//     PlcTask Inputs/GVL_iXlinker.EtherCAT_Master_ERxxxx.Beckhoff_ER2xxx.Beckhoff_ER2xxxEK1122.A_0015_ER2038_0002_0018.Diag_Channel_4.Input <-> Diag Channel 4/Input
//     PlcTask Inputs/GVL_iXlinker.EtherCAT_Master_ERxxxx.Beckhoff_ER2xxx.Beckhoff_ER2xxxEK1122.A_0015_ER2038_0002_0018.Diag_Channel_5.Input <-> Diag Channel 5/Input
//     PlcTask Inputs/GVL_iXlinker.EtherCAT_Master_ERxxxx.Beckhoff_ER2xxx.Beckhoff_ER2xxxEK1122.A_0015_ER2038_0002_0018.Diag_Channel_6.Input <-> Diag Channel 6/Input
//     PlcTask Inputs/GVL_iXlinker.EtherCAT_Master_ERxxxx.Beckhoff_ER2xxx.Beckhoff_ER2xxxEK1122.A_0015_ER2038_0002_0018.Diag_Channel_7.Input <-> Diag Channel 7/Input
//     PlcTask Inputs/GVL_iXlinker.EtherCAT_Master_ERxxxx.Beckhoff_ER2xxx.Beckhoff_ER2xxxEK1122.A_0015_ER2038_0002_0018.Diag_Channel_8.Input <-> Diag Channel 8/Input
//     PlcTask Outputs/GVL_iXlinker.EtherCAT_Master_ERxxxx.Beckhoff_ER2xxx.Beckhoff_ER2xxxEK1122.A_0015_ER2038_0002_0018.Channel_1.Output <-> Channel 1/Output
//     PlcTask Outputs/GVL_iXlinker.EtherCAT_Master_ERxxxx.Beckhoff_ER2xxx.Beckhoff_ER2xxxEK1122.A_0015_ER2038_0002_0018.Channel_2.Output <-> Channel 2/Output
//     PlcTask Outputs/GVL_iXlinker.EtherCAT_Master_ERxxxx.Beckhoff_ER2xxx.Beckhoff_ER2xxxEK1122.A_0015_ER2038_0002_0018.Channel_3.Output <-> Channel 3/Output
//     PlcTask Outputs/GVL_iXlinker.EtherCAT_Master_ERxxxx.Beckhoff_ER2xxx.Beckhoff_ER2xxxEK1122.A_0015_ER2038_0002_0018.Channel_4.Output <-> Channel 4/Output
//     PlcTask Outputs/GVL_iXlinker.EtherCAT_Master_ERxxxx.Beckhoff_ER2xxx.Beckhoff_ER2xxxEK1122.A_0015_ER2038_0002_0018.Channel_5.Output <-> Channel 5/Output
//     PlcTask Outputs/GVL_iXlinker.EtherCAT_Master_ERxxxx.Beckhoff_ER2xxx.Beckhoff_ER2xxxEK1122.A_0015_ER2038_0002_0018.Channel_6.Output <-> Channel 6/Output
//     PlcTask Outputs/GVL_iXlinker.EtherCAT_Master_ERxxxx.Beckhoff_ER2xxx.Beckhoff_ER2xxxEK1122.A_0015_ER2038_0002_0018.Channel_7.Output <-> Channel 7/Output
//     PlcTask Outputs/GVL_iXlinker.EtherCAT_Master_ERxxxx.Beckhoff_ER2xxx.Beckhoff_ER2xxxEK1122.A_0015_ER2038_0002_0018.Channel_8.Output <-> Channel 8/Output
//     PlcTask Inputs/GVL_iXlinker.EtherCAT_Master_ERxxxx.Beckhoff_ER2xxx.Beckhoff_ER2xxxEK1122.A_0015_ER2038_0002_0018.WcState.WcState <-> WcState/WcState
//     PlcTask Inputs/GVL_iXlinker.EtherCAT_Master_ERxxxx.Beckhoff_ER2xxx.Beckhoff_ER2xxxEK1122.A_0015_ER2038_0002_0018.WcState.InputToggle <-> WcState/InputToggle
//     PlcTask Inputs/GVL_iXlinker.EtherCAT_Master_ERxxxx.Beckhoff_ER2xxx.Beckhoff_ER2xxxEK1122.A_0015_ER2038_0002_0018.InfoData.State <-> InfoData/State
//   PLC/PLC Instance <-> EtherCAT Master ERxxxx/Beckhoff ER2xxx/Beckhoff ER2xxxEK1122/A_0016(ER2308-0001-0018)
//     PlcTask Inputs/GVL_iXlinker.EtherCAT_Master_ERxxxx.Beckhoff_ER2xxx.Beckhoff_ER2xxxEK1122.A_0016_ER2308_0001_0018.Channel_1.Input <-> Channel 1/Input
//     PlcTask Inputs/GVL_iXlinker.EtherCAT_Master_ERxxxx.Beckhoff_ER2xxx.Beckhoff_ER2xxxEK1122.A_0016_ER2308_0001_0018.Channel_2.Input <-> Channel 2/Input
//     PlcTask Inputs/GVL_iXlinker.EtherCAT_Master_ERxxxx.Beckhoff_ER2xxx.Beckhoff_ER2xxxEK1122.A_0016_ER2308_0001_0018.Channel_3.Input <-> Channel 3/Input
//     PlcTask Inputs/GVL_iXlinker.EtherCAT_Master_ERxxxx.Beckhoff_ER2xxx.Beckhoff_ER2xxxEK1122.A_0016_ER2308_0001_0018.Channel_4.Input <-> Channel 4/Input
//     PlcTask Outputs/GVL_iXlinker.EtherCAT_Master_ERxxxx.Beckhoff_ER2xxx.Beckhoff_ER2xxxEK1122.A_0016_ER2308_0001_0018.Channel_5.Output <-> Channel 5/Output
//     PlcTask Outputs/GVL_iXlinker.EtherCAT_Master_ERxxxx.Beckhoff_ER2xxx.Beckhoff_ER2xxxEK1122.A_0016_ER2308_0001_0018.Channel_6.Output <-> Channel 6/Output
//     PlcTask Outputs/GVL_iXlinker.EtherCAT_Master_ERxxxx.Beckhoff_ER2xxx.Beckhoff_ER2xxxEK1122.A_0016_ER2308_0001_0018.Channel_7.Output <-> Channel 7/Output
//     PlcTask Outputs/GVL_iXlinker.EtherCAT_Master_ERxxxx.Beckhoff_ER2xxx.Beckhoff_ER2xxxEK1122.A_0016_ER2308_0001_0018.Channel_8.Output <-> Channel 8/Output
//     PlcTask Inputs/GVL_iXlinker.EtherCAT_Master_ERxxxx.Beckhoff_ER2xxx.Beckhoff_ER2xxxEK1122.A_0016_ER2308_0001_0018.WcState.WcState <-> WcState/WcState
//     PlcTask Inputs/GVL_iXlinker.EtherCAT_Master_ERxxxx.Beckhoff_ER2xxx.Beckhoff_ER2xxxEK1122.A_0016_ER2308_0001_0018.WcState.InputToggle <-> WcState/InputToggle
//     PlcTask Inputs/GVL_iXlinker.EtherCAT_Master_ERxxxx.Beckhoff_ER2xxx.Beckhoff_ER2xxxEK1122.A_0016_ER2308_0001_0018.InfoData.State <-> InfoData/State
//   PLC/PLC Instance <-> EtherCAT Master ERxxxx/Beckhoff ER2xxx/Beckhoff ER2xxxEK1122/A_0017(ER2308-0001-0019)
//     PlcTask Inputs/GVL_iXlinker.EtherCAT_Master_ERxxxx.Beckhoff_ER2xxx.Beckhoff_ER2xxxEK1122.A_0017_ER2308_0001_0019.Channel_1.Input <-> Channel 1/Input
//     PlcTask Inputs/GVL_iXlinker.EtherCAT_Master_ERxxxx.Beckhoff_ER2xxx.Beckhoff_ER2xxxEK1122.A_0017_ER2308_0001_0019.Channel_2.Input <-> Channel 2/Input
//     PlcTask Inputs/GVL_iXlinker.EtherCAT_Master_ERxxxx.Beckhoff_ER2xxx.Beckhoff_ER2xxxEK1122.A_0017_ER2308_0001_0019.Channel_3.Input <-> Channel 3/Input
//     PlcTask Inputs/GVL_iXlinker.EtherCAT_Master_ERxxxx.Beckhoff_ER2xxx.Beckhoff_ER2xxxEK1122.A_0017_ER2308_0001_0019.Channel_4.Input <-> Channel 4/Input
//     PlcTask Outputs/GVL_iXlinker.EtherCAT_Master_ERxxxx.Beckhoff_ER2xxx.Beckhoff_ER2xxxEK1122.A_0017_ER2308_0001_0019.Channel_5.Output <-> Channel 5/Output
//     PlcTask Outputs/GVL_iXlinker.EtherCAT_Master_ERxxxx.Beckhoff_ER2xxx.Beckhoff_ER2xxxEK1122.A_0017_ER2308_0001_0019.Channel_6.Output <-> Channel 6/Output
//     PlcTask Outputs/GVL_iXlinker.EtherCAT_Master_ERxxxx.Beckhoff_ER2xxx.Beckhoff_ER2xxxEK1122.A_0017_ER2308_0001_0019.Channel_7.Output <-> Channel 7/Output
//     PlcTask Outputs/GVL_iXlinker.EtherCAT_Master_ERxxxx.Beckhoff_ER2xxx.Beckhoff_ER2xxxEK1122.A_0017_ER2308_0001_0019.Channel_8.Output <-> Channel 8/Output
//     PlcTask Inputs/GVL_iXlinker.EtherCAT_Master_ERxxxx.Beckhoff_ER2xxx.Beckhoff_ER2xxxEK1122.A_0017_ER2308_0001_0019.WcState.WcState <-> WcState/WcState
//     PlcTask Inputs/GVL_iXlinker.EtherCAT_Master_ERxxxx.Beckhoff_ER2xxx.Beckhoff_ER2xxxEK1122.A_0017_ER2308_0001_0019.WcState.InputToggle <-> WcState/InputToggle
//     PlcTask Inputs/GVL_iXlinker.EtherCAT_Master_ERxxxx.Beckhoff_ER2xxx.Beckhoff_ER2xxxEK1122.A_0017_ER2308_0001_0019.InfoData.State <-> InfoData/State
//   PLC/PLC Instance <-> EtherCAT Master ERxxxx/Beckhoff ER2xxx/Beckhoff ER2xxxEK1122/A_0018(ER2308-0002-0018)
//     PlcTask Inputs/GVL_iXlinker.EtherCAT_Master_ERxxxx.Beckhoff_ER2xxx.Beckhoff_ER2xxxEK1122.A_0018_ER2308_0002_0018.Channel_1.Input <-> Channel 1/Input
//     PlcTask Inputs/GVL_iXlinker.EtherCAT_Master_ERxxxx.Beckhoff_ER2xxx.Beckhoff_ER2xxxEK1122.A_0018_ER2308_0002_0018.Channel_2.Input <-> Channel 2/Input
//     PlcTask Inputs/GVL_iXlinker.EtherCAT_Master_ERxxxx.Beckhoff_ER2xxx.Beckhoff_ER2xxxEK1122.A_0018_ER2308_0002_0018.Channel_3.Input <-> Channel 3/Input
//     PlcTask Inputs/GVL_iXlinker.EtherCAT_Master_ERxxxx.Beckhoff_ER2xxx.Beckhoff_ER2xxxEK1122.A_0018_ER2308_0002_0018.Channel_4.Input <-> Channel 4/Input
//     PlcTask Outputs/GVL_iXlinker.EtherCAT_Master_ERxxxx.Beckhoff_ER2xxx.Beckhoff_ER2xxxEK1122.A_0018_ER2308_0002_0018.Channel_5.Output <-> Channel 5/Output
//     PlcTask Outputs/GVL_iXlinker.EtherCAT_Master_ERxxxx.Beckhoff_ER2xxx.Beckhoff_ER2xxxEK1122.A_0018_ER2308_0002_0018.Channel_6.Output <-> Channel 6/Output
//     PlcTask Outputs/GVL_iXlinker.EtherCAT_Master_ERxxxx.Beckhoff_ER2xxx.Beckhoff_ER2xxxEK1122.A_0018_ER2308_0002_0018.Channel_7.Output <-> Channel 7/Output
//     PlcTask Outputs/GVL_iXlinker.EtherCAT_Master_ERxxxx.Beckhoff_ER2xxx.Beckhoff_ER2xxxEK1122.A_0018_ER2308_0002_0018.Channel_8.Output <-> Channel 8/Output
//     PlcTask Inputs/GVL_iXlinker.EtherCAT_Master_ERxxxx.Beckhoff_ER2xxx.Beckhoff_ER2xxxEK1122.A_0018_ER2308_0002_0018.WcState.WcState <-> WcState/WcState
//     PlcTask Inputs/GVL_iXlinker.EtherCAT_Master_ERxxxx.Beckhoff_ER2xxx.Beckhoff_ER2xxxEK1122.A_0018_ER2308_0002_0018.WcState.InputToggle <-> WcState/InputToggle
//     PlcTask Inputs/GVL_iXlinker.EtherCAT_Master_ERxxxx.Beckhoff_ER2xxx.Beckhoff_ER2xxxEK1122.A_0018_ER2308_0002_0018.InfoData.State <-> InfoData/State
//   PLC/PLC Instance <-> EtherCAT Master ERxxxx/Beckhoff ER2xxx/Beckhoff ER2xxxEK1122/A_0019(ER2308-0002-0019)
//     PlcTask Inputs/GVL_iXlinker.EtherCAT_Master_ERxxxx.Beckhoff_ER2xxx.Beckhoff_ER2xxxEK1122.A_0019_ER2308_0002_0019.Channel_1.Input <-> Channel 1/Input
//     PlcTask Inputs/GVL_iXlinker.EtherCAT_Master_ERxxxx.Beckhoff_ER2xxx.Beckhoff_ER2xxxEK1122.A_0019_ER2308_0002_0019.Channel_2.Input <-> Channel 2/Input
//     PlcTask Inputs/GVL_iXlinker.EtherCAT_Master_ERxxxx.Beckhoff_ER2xxx.Beckhoff_ER2xxxEK1122.A_0019_ER2308_0002_0019.Channel_3.Input <-> Channel 3/Input
//     PlcTask Inputs/GVL_iXlinker.EtherCAT_Master_ERxxxx.Beckhoff_ER2xxx.Beckhoff_ER2xxxEK1122.A_0019_ER2308_0002_0019.Channel_4.Input <-> Channel 4/Input
//     PlcTask Outputs/GVL_iXlinker.EtherCAT_Master_ERxxxx.Beckhoff_ER2xxx.Beckhoff_ER2xxxEK1122.A_0019_ER2308_0002_0019.Channel_5.Output <-> Channel 5/Output
//     PlcTask Outputs/GVL_iXlinker.EtherCAT_Master_ERxxxx.Beckhoff_ER2xxx.Beckhoff_ER2xxxEK1122.A_0019_ER2308_0002_0019.Channel_6.Output <-> Channel 6/Output
//     PlcTask Outputs/GVL_iXlinker.EtherCAT_Master_ERxxxx.Beckhoff_ER2xxx.Beckhoff_ER2xxxEK1122.A_0019_ER2308_0002_0019.Channel_7.Output <-> Channel 7/Output
//     PlcTask Outputs/GVL_iXlinker.EtherCAT_Master_ERxxxx.Beckhoff_ER2xxx.Beckhoff_ER2xxxEK1122.A_0019_ER2308_0002_0019.Channel_8.Output <-> Channel 8/Output
//     PlcTask Inputs/GVL_iXlinker.EtherCAT_Master_ERxxxx.Beckhoff_ER2xxx.Beckhoff_ER2xxxEK1122.A_0019_ER2308_0002_0019.WcState.WcState <-> WcState/WcState
//     PlcTask Inputs/GVL_iXlinker.EtherCAT_Master_ERxxxx.Beckhoff_ER2xxx.Beckhoff_ER2xxxEK1122.A_0019_ER2308_0002_0019.WcState.InputToggle <-> WcState/InputToggle
//     PlcTask Inputs/GVL_iXlinker.EtherCAT_Master_ERxxxx.Beckhoff_ER2xxx.Beckhoff_ER2xxxEK1122.A_0019_ER2308_0002_0019.InfoData.State <-> InfoData/State
//   PLC/PLC Instance <-> EtherCAT Master ERxxxx/Beckhoff ER2xxx/Beckhoff ER2xxxEK1122/A_0020(ER2318-0001-0018)
//     PlcTask Inputs/GVL_iXlinker.EtherCAT_Master_ERxxxx.Beckhoff_ER2xxx.Beckhoff_ER2xxxEK1122.A_0020_ER2318_0001_0018.Channel_1.Input <-> Channel 1/Input
//     PlcTask Inputs/GVL_iXlinker.EtherCAT_Master_ERxxxx.Beckhoff_ER2xxx.Beckhoff_ER2xxxEK1122.A_0020_ER2318_0001_0018.Channel_2.Input <-> Channel 2/Input
//     PlcTask Inputs/GVL_iXlinker.EtherCAT_Master_ERxxxx.Beckhoff_ER2xxx.Beckhoff_ER2xxxEK1122.A_0020_ER2318_0001_0018.Channel_3.Input <-> Channel 3/Input
//     PlcTask Inputs/GVL_iXlinker.EtherCAT_Master_ERxxxx.Beckhoff_ER2xxx.Beckhoff_ER2xxxEK1122.A_0020_ER2318_0001_0018.Channel_4.Input <-> Channel 4/Input
//     PlcTask Outputs/GVL_iXlinker.EtherCAT_Master_ERxxxx.Beckhoff_ER2xxx.Beckhoff_ER2xxxEK1122.A_0020_ER2318_0001_0018.Channel_5.Output <-> Channel 5/Output
//     PlcTask Outputs/GVL_iXlinker.EtherCAT_Master_ERxxxx.Beckhoff_ER2xxx.Beckhoff_ER2xxxEK1122.A_0020_ER2318_0001_0018.Channel_6.Output <-> Channel 6/Output
//     PlcTask Outputs/GVL_iXlinker.EtherCAT_Master_ERxxxx.Beckhoff_ER2xxx.Beckhoff_ER2xxxEK1122.A_0020_ER2318_0001_0018.Channel_7.Output <-> Channel 7/Output
//     PlcTask Outputs/GVL_iXlinker.EtherCAT_Master_ERxxxx.Beckhoff_ER2xxx.Beckhoff_ER2xxxEK1122.A_0020_ER2318_0001_0018.Channel_8.Output <-> Channel 8/Output
//     PlcTask Inputs/GVL_iXlinker.EtherCAT_Master_ERxxxx.Beckhoff_ER2xxx.Beckhoff_ER2xxxEK1122.A_0020_ER2318_0001_0018.WcState.WcState <-> WcState/WcState
//     PlcTask Inputs/GVL_iXlinker.EtherCAT_Master_ERxxxx.Beckhoff_ER2xxx.Beckhoff_ER2xxxEK1122.A_0020_ER2318_0001_0018.WcState.InputToggle <-> WcState/InputToggle
//     PlcTask Inputs/GVL_iXlinker.EtherCAT_Master_ERxxxx.Beckhoff_ER2xxx.Beckhoff_ER2xxxEK1122.A_0020_ER2318_0001_0018.InfoData.State <-> InfoData/State
//   PLC/PLC Instance <-> EtherCAT Master ERxxxx/Beckhoff ER2xxx/Beckhoff ER2xxxEK1122/A_0021(ER2318-0001-0019)
//     PlcTask Inputs/GVL_iXlinker.EtherCAT_Master_ERxxxx.Beckhoff_ER2xxx.Beckhoff_ER2xxxEK1122.A_0021_ER2318_0001_0019.Channel_1.Input <-> Channel 1/Input
//     PlcTask Inputs/GVL_iXlinker.EtherCAT_Master_ERxxxx.Beckhoff_ER2xxx.Beckhoff_ER2xxxEK1122.A_0021_ER2318_0001_0019.Channel_2.Input <-> Channel 2/Input
//     PlcTask Inputs/GVL_iXlinker.EtherCAT_Master_ERxxxx.Beckhoff_ER2xxx.Beckhoff_ER2xxxEK1122.A_0021_ER2318_0001_0019.Channel_3.Input <-> Channel 3/Input
//     PlcTask Inputs/GVL_iXlinker.EtherCAT_Master_ERxxxx.Beckhoff_ER2xxx.Beckhoff_ER2xxxEK1122.A_0021_ER2318_0001_0019.Channel_4.Input <-> Channel 4/Input
//     PlcTask Outputs/GVL_iXlinker.EtherCAT_Master_ERxxxx.Beckhoff_ER2xxx.Beckhoff_ER2xxxEK1122.A_0021_ER2318_0001_0019.Channel_5.Output <-> Channel 5/Output
//     PlcTask Outputs/GVL_iXlinker.EtherCAT_Master_ERxxxx.Beckhoff_ER2xxx.Beckhoff_ER2xxxEK1122.A_0021_ER2318_0001_0019.Channel_6.Output <-> Channel 6/Output
//     PlcTask Outputs/GVL_iXlinker.EtherCAT_Master_ERxxxx.Beckhoff_ER2xxx.Beckhoff_ER2xxxEK1122.A_0021_ER2318_0001_0019.Channel_7.Output <-> Channel 7/Output
//     PlcTask Outputs/GVL_iXlinker.EtherCAT_Master_ERxxxx.Beckhoff_ER2xxx.Beckhoff_ER2xxxEK1122.A_0021_ER2318_0001_0019.Channel_8.Output <-> Channel 8/Output
//     PlcTask Inputs/GVL_iXlinker.EtherCAT_Master_ERxxxx.Beckhoff_ER2xxx.Beckhoff_ER2xxxEK1122.A_0021_ER2318_0001_0019.WcState.WcState <-> WcState/WcState
//     PlcTask Inputs/GVL_iXlinker.EtherCAT_Master_ERxxxx.Beckhoff_ER2xxx.Beckhoff_ER2xxxEK1122.A_0021_ER2318_0001_0019.WcState.InputToggle <-> WcState/InputToggle
//     PlcTask Inputs/GVL_iXlinker.EtherCAT_Master_ERxxxx.Beckhoff_ER2xxx.Beckhoff_ER2xxxEK1122.A_0021_ER2318_0001_0019.InfoData.State <-> InfoData/State
//   PLC/PLC Instance <-> EtherCAT Master ERxxxx/Beckhoff ER2xxx/Beckhoff ER2xxxEK1122/A_0022(ER2318-0002-0018)
//     PlcTask Inputs/GVL_iXlinker.EtherCAT_Master_ERxxxx.Beckhoff_ER2xxx.Beckhoff_ER2xxxEK1122.A_0022_ER2318_0002_0018.Channel_1.Input <-> Channel 1/Input
//     PlcTask Inputs/GVL_iXlinker.EtherCAT_Master_ERxxxx.Beckhoff_ER2xxx.Beckhoff_ER2xxxEK1122.A_0022_ER2318_0002_0018.Channel_2.Input <-> Channel 2/Input
//     PlcTask Inputs/GVL_iXlinker.EtherCAT_Master_ERxxxx.Beckhoff_ER2xxx.Beckhoff_ER2xxxEK1122.A_0022_ER2318_0002_0018.Channel_3.Input <-> Channel 3/Input
//     PlcTask Inputs/GVL_iXlinker.EtherCAT_Master_ERxxxx.Beckhoff_ER2xxx.Beckhoff_ER2xxxEK1122.A_0022_ER2318_0002_0018.Channel_4.Input <-> Channel 4/Input
//     PlcTask Outputs/GVL_iXlinker.EtherCAT_Master_ERxxxx.Beckhoff_ER2xxx.Beckhoff_ER2xxxEK1122.A_0022_ER2318_0002_0018.Channel_5.Output <-> Channel 5/Output
//     PlcTask Outputs/GVL_iXlinker.EtherCAT_Master_ERxxxx.Beckhoff_ER2xxx.Beckhoff_ER2xxxEK1122.A_0022_ER2318_0002_0018.Channel_6.Output <-> Channel 6/Output
//     PlcTask Outputs/GVL_iXlinker.EtherCAT_Master_ERxxxx.Beckhoff_ER2xxx.Beckhoff_ER2xxxEK1122.A_0022_ER2318_0002_0018.Channel_7.Output <-> Channel 7/Output
//     PlcTask Outputs/GVL_iXlinker.EtherCAT_Master_ERxxxx.Beckhoff_ER2xxx.Beckhoff_ER2xxxEK1122.A_0022_ER2318_0002_0018.Channel_8.Output <-> Channel 8/Output
//     PlcTask Inputs/GVL_iXlinker.EtherCAT_Master_ERxxxx.Beckhoff_ER2xxx.Beckhoff_ER2xxxEK1122.A_0022_ER2318_0002_0018.WcState.WcState <-> WcState/WcState
//     PlcTask Inputs/GVL_iXlinker.EtherCAT_Master_ERxxxx.Beckhoff_ER2xxx.Beckhoff_ER2xxxEK1122.A_0022_ER2318_0002_0018.WcState.InputToggle <-> WcState/InputToggle
//     PlcTask Inputs/GVL_iXlinker.EtherCAT_Master_ERxxxx.Beckhoff_ER2xxx.Beckhoff_ER2xxxEK1122.A_0022_ER2318_0002_0018.InfoData.State <-> InfoData/State
//   PLC/PLC Instance <-> EtherCAT Master ERxxxx/Beckhoff ER2xxx/Beckhoff ER2xxxEK1122/A_0023(ER2318-0002-0019)
//     PlcTask Inputs/GVL_iXlinker.EtherCAT_Master_ERxxxx.Beckhoff_ER2xxx.Beckhoff_ER2xxxEK1122.A_0023_ER2318_0002_0019.Channel_1.Input <-> Channel 1/Input
//     PlcTask Inputs/GVL_iXlinker.EtherCAT_Master_ERxxxx.Beckhoff_ER2xxx.Beckhoff_ER2xxxEK1122.A_0023_ER2318_0002_0019.Channel_2.Input <-> Channel 2/Input
//     PlcTask Inputs/GVL_iXlinker.EtherCAT_Master_ERxxxx.Beckhoff_ER2xxx.Beckhoff_ER2xxxEK1122.A_0023_ER2318_0002_0019.Channel_3.Input <-> Channel 3/Input
//     PlcTask Inputs/GVL_iXlinker.EtherCAT_Master_ERxxxx.Beckhoff_ER2xxx.Beckhoff_ER2xxxEK1122.A_0023_ER2318_0002_0019.Channel_4.Input <-> Channel 4/Input
//     PlcTask Outputs/GVL_iXlinker.EtherCAT_Master_ERxxxx.Beckhoff_ER2xxx.Beckhoff_ER2xxxEK1122.A_0023_ER2318_0002_0019.Channel_5.Output <-> Channel 5/Output
//     PlcTask Outputs/GVL_iXlinker.EtherCAT_Master_ERxxxx.Beckhoff_ER2xxx.Beckhoff_ER2xxxEK1122.A_0023_ER2318_0002_0019.Channel_6.Output <-> Channel 6/Output
//     PlcTask Outputs/GVL_iXlinker.EtherCAT_Master_ERxxxx.Beckhoff_ER2xxx.Beckhoff_ER2xxxEK1122.A_0023_ER2318_0002_0019.Channel_7.Output <-> Channel 7/Output
//     PlcTask Outputs/GVL_iXlinker.EtherCAT_Master_ERxxxx.Beckhoff_ER2xxx.Beckhoff_ER2xxxEK1122.A_0023_ER2318_0002_0019.Channel_8.Output <-> Channel 8/Output
//     PlcTask Inputs/GVL_iXlinker.EtherCAT_Master_ERxxxx.Beckhoff_ER2xxx.Beckhoff_ER2xxxEK1122.A_0023_ER2318_0002_0019.WcState.WcState <-> WcState/WcState
//     PlcTask Inputs/GVL_iXlinker.EtherCAT_Master_ERxxxx.Beckhoff_ER2xxx.Beckhoff_ER2xxxEK1122.A_0023_ER2318_0002_0019.WcState.InputToggle <-> WcState/InputToggle
//     PlcTask Inputs/GVL_iXlinker.EtherCAT_Master_ERxxxx.Beckhoff_ER2xxx.Beckhoff_ER2xxxEK1122.A_0023_ER2318_0002_0019.InfoData.State <-> InfoData/State
//   PLC/PLC Instance <-> EtherCAT Master ERxxxx/Beckhoff ER2xxx/Beckhoff ER2xxxEK1122/A_0024(ER2328-0001-0017)
//     PlcTask Inputs/GVL_iXlinker.EtherCAT_Master_ERxxxx.Beckhoff_ER2xxx.Beckhoff_ER2xxxEK1122.A_0024_ER2328_0001_0017.Channel_1.Input <-> Channel 1/Input
//     PlcTask Inputs/GVL_iXlinker.EtherCAT_Master_ERxxxx.Beckhoff_ER2xxx.Beckhoff_ER2xxxEK1122.A_0024_ER2328_0001_0017.Channel_2.Input <-> Channel 2/Input
//     PlcTask Inputs/GVL_iXlinker.EtherCAT_Master_ERxxxx.Beckhoff_ER2xxx.Beckhoff_ER2xxxEK1122.A_0024_ER2328_0001_0017.Channel_3.Input <-> Channel 3/Input
//     PlcTask Inputs/GVL_iXlinker.EtherCAT_Master_ERxxxx.Beckhoff_ER2xxx.Beckhoff_ER2xxxEK1122.A_0024_ER2328_0001_0017.Channel_4.Input <-> Channel 4/Input
//     PlcTask Outputs/GVL_iXlinker.EtherCAT_Master_ERxxxx.Beckhoff_ER2xxx.Beckhoff_ER2xxxEK1122.A_0024_ER2328_0001_0017.Channel_5.Output <-> Channel 5/Output
//     PlcTask Outputs/GVL_iXlinker.EtherCAT_Master_ERxxxx.Beckhoff_ER2xxx.Beckhoff_ER2xxxEK1122.A_0024_ER2328_0001_0017.Channel_6.Output <-> Channel 6/Output
//     PlcTask Outputs/GVL_iXlinker.EtherCAT_Master_ERxxxx.Beckhoff_ER2xxx.Beckhoff_ER2xxxEK1122.A_0024_ER2328_0001_0017.Channel_7.Output <-> Channel 7/Output
//     PlcTask Outputs/GVL_iXlinker.EtherCAT_Master_ERxxxx.Beckhoff_ER2xxx.Beckhoff_ER2xxxEK1122.A_0024_ER2328_0001_0017.Channel_8.Output <-> Channel 8/Output
//     PlcTask Inputs/GVL_iXlinker.EtherCAT_Master_ERxxxx.Beckhoff_ER2xxx.Beckhoff_ER2xxxEK1122.A_0024_ER2328_0001_0017.WcState.WcState <-> WcState/WcState
//     PlcTask Inputs/GVL_iXlinker.EtherCAT_Master_ERxxxx.Beckhoff_ER2xxx.Beckhoff_ER2xxxEK1122.A_0024_ER2328_0001_0017.WcState.InputToggle <-> WcState/InputToggle
//     PlcTask Inputs/GVL_iXlinker.EtherCAT_Master_ERxxxx.Beckhoff_ER2xxx.Beckhoff_ER2xxxEK1122.A_0024_ER2328_0001_0017.InfoData.State <-> InfoData/State
//   PLC/PLC Instance <-> EtherCAT Master ERxxxx/Beckhoff ER2xxx/Beckhoff ER2xxxEK1122/A_0025(ER2328-0001-0018)
//     PlcTask Inputs/GVL_iXlinker.EtherCAT_Master_ERxxxx.Beckhoff_ER2xxx.Beckhoff_ER2xxxEK1122.A_0025_ER2328_0001_0018.Channel_1.Input <-> Channel 1/Input
//     PlcTask Inputs/GVL_iXlinker.EtherCAT_Master_ERxxxx.Beckhoff_ER2xxx.Beckhoff_ER2xxxEK1122.A_0025_ER2328_0001_0018.Channel_2.Input <-> Channel 2/Input
//     PlcTask Inputs/GVL_iXlinker.EtherCAT_Master_ERxxxx.Beckhoff_ER2xxx.Beckhoff_ER2xxxEK1122.A_0025_ER2328_0001_0018.Channel_3.Input <-> Channel 3/Input
//     PlcTask Inputs/GVL_iXlinker.EtherCAT_Master_ERxxxx.Beckhoff_ER2xxx.Beckhoff_ER2xxxEK1122.A_0025_ER2328_0001_0018.Channel_4.Input <-> Channel 4/Input
//     PlcTask Outputs/GVL_iXlinker.EtherCAT_Master_ERxxxx.Beckhoff_ER2xxx.Beckhoff_ER2xxxEK1122.A_0025_ER2328_0001_0018.Channel_5.Output <-> Channel 5/Output
//     PlcTask Outputs/GVL_iXlinker.EtherCAT_Master_ERxxxx.Beckhoff_ER2xxx.Beckhoff_ER2xxxEK1122.A_0025_ER2328_0001_0018.Channel_6.Output <-> Channel 6/Output
//     PlcTask Outputs/GVL_iXlinker.EtherCAT_Master_ERxxxx.Beckhoff_ER2xxx.Beckhoff_ER2xxxEK1122.A_0025_ER2328_0001_0018.Channel_7.Output <-> Channel 7/Output
//     PlcTask Outputs/GVL_iXlinker.EtherCAT_Master_ERxxxx.Beckhoff_ER2xxx.Beckhoff_ER2xxxEK1122.A_0025_ER2328_0001_0018.Channel_8.Output <-> Channel 8/Output
//     PlcTask Inputs/GVL_iXlinker.EtherCAT_Master_ERxxxx.Beckhoff_ER2xxx.Beckhoff_ER2xxxEK1122.A_0025_ER2328_0001_0018.WcState.WcState <-> WcState/WcState
//     PlcTask Inputs/GVL_iXlinker.EtherCAT_Master_ERxxxx.Beckhoff_ER2xxx.Beckhoff_ER2xxxEK1122.A_0025_ER2328_0001_0018.WcState.InputToggle <-> WcState/InputToggle
//     PlcTask Inputs/GVL_iXlinker.EtherCAT_Master_ERxxxx.Beckhoff_ER2xxx.Beckhoff_ER2xxxEK1122.A_0025_ER2328_0001_0018.InfoData.State <-> InfoData/State
//   PLC/PLC Instance <-> EtherCAT Master ERxxxx/Beckhoff ER2xxx/Beckhoff ER2xxxEK1122/A_0026(ER2328-0002-0018)
//     PlcTask Inputs/GVL_iXlinker.EtherCAT_Master_ERxxxx.Beckhoff_ER2xxx.Beckhoff_ER2xxxEK1122.A_0026_ER2328_0002_0018.Channel_1.Input <-> Channel 1/Input
//     PlcTask Inputs/GVL_iXlinker.EtherCAT_Master_ERxxxx.Beckhoff_ER2xxx.Beckhoff_ER2xxxEK1122.A_0026_ER2328_0002_0018.Channel_2.Input <-> Channel 2/Input
//     PlcTask Inputs/GVL_iXlinker.EtherCAT_Master_ERxxxx.Beckhoff_ER2xxx.Beckhoff_ER2xxxEK1122.A_0026_ER2328_0002_0018.Channel_3.Input <-> Channel 3/Input
//     PlcTask Inputs/GVL_iXlinker.EtherCAT_Master_ERxxxx.Beckhoff_ER2xxx.Beckhoff_ER2xxxEK1122.A_0026_ER2328_0002_0018.Channel_4.Input <-> Channel 4/Input
//     PlcTask Outputs/GVL_iXlinker.EtherCAT_Master_ERxxxx.Beckhoff_ER2xxx.Beckhoff_ER2xxxEK1122.A_0026_ER2328_0002_0018.Channel_5.Output <-> Channel 5/Output
//     PlcTask Outputs/GVL_iXlinker.EtherCAT_Master_ERxxxx.Beckhoff_ER2xxx.Beckhoff_ER2xxxEK1122.A_0026_ER2328_0002_0018.Channel_6.Output <-> Channel 6/Output
//     PlcTask Outputs/GVL_iXlinker.EtherCAT_Master_ERxxxx.Beckhoff_ER2xxx.Beckhoff_ER2xxxEK1122.A_0026_ER2328_0002_0018.Channel_7.Output <-> Channel 7/Output
//     PlcTask Outputs/GVL_iXlinker.EtherCAT_Master_ERxxxx.Beckhoff_ER2xxx.Beckhoff_ER2xxxEK1122.A_0026_ER2328_0002_0018.Channel_8.Output <-> Channel 8/Output
//     PlcTask Inputs/GVL_iXlinker.EtherCAT_Master_ERxxxx.Beckhoff_ER2xxx.Beckhoff_ER2xxxEK1122.A_0026_ER2328_0002_0018.WcState.WcState <-> WcState/WcState
//     PlcTask Inputs/GVL_iXlinker.EtherCAT_Master_ERxxxx.Beckhoff_ER2xxx.Beckhoff_ER2xxxEK1122.A_0026_ER2328_0002_0018.WcState.InputToggle <-> WcState/InputToggle
//     PlcTask Inputs/GVL_iXlinker.EtherCAT_Master_ERxxxx.Beckhoff_ER2xxx.Beckhoff_ER2xxxEK1122.A_0026_ER2328_0002_0018.InfoData.State <-> InfoData/State
//   PLC/PLC Instance <-> EtherCAT Master ERxxxx/Beckhoff ER2xxx/Beckhoff ER2xxxEK1122/A_0027(ER2328-0002-0019)
//     PlcTask Inputs/GVL_iXlinker.EtherCAT_Master_ERxxxx.Beckhoff_ER2xxx.Beckhoff_ER2xxxEK1122.A_0027_ER2328_0002_0019.Channel_1.Input <-> Channel 1/Input
//     PlcTask Inputs/GVL_iXlinker.EtherCAT_Master_ERxxxx.Beckhoff_ER2xxx.Beckhoff_ER2xxxEK1122.A_0027_ER2328_0002_0019.Channel_2.Input <-> Channel 2/Input
//     PlcTask Inputs/GVL_iXlinker.EtherCAT_Master_ERxxxx.Beckhoff_ER2xxx.Beckhoff_ER2xxxEK1122.A_0027_ER2328_0002_0019.Channel_3.Input <-> Channel 3/Input
//     PlcTask Inputs/GVL_iXlinker.EtherCAT_Master_ERxxxx.Beckhoff_ER2xxx.Beckhoff_ER2xxxEK1122.A_0027_ER2328_0002_0019.Channel_4.Input <-> Channel 4/Input
//     PlcTask Outputs/GVL_iXlinker.EtherCAT_Master_ERxxxx.Beckhoff_ER2xxx.Beckhoff_ER2xxxEK1122.A_0027_ER2328_0002_0019.Channel_5.Output <-> Channel 5/Output
//     PlcTask Outputs/GVL_iXlinker.EtherCAT_Master_ERxxxx.Beckhoff_ER2xxx.Beckhoff_ER2xxxEK1122.A_0027_ER2328_0002_0019.Channel_6.Output <-> Channel 6/Output
//     PlcTask Outputs/GVL_iXlinker.EtherCAT_Master_ERxxxx.Beckhoff_ER2xxx.Beckhoff_ER2xxxEK1122.A_0027_ER2328_0002_0019.Channel_7.Output <-> Channel 7/Output
//     PlcTask Outputs/GVL_iXlinker.EtherCAT_Master_ERxxxx.Beckhoff_ER2xxx.Beckhoff_ER2xxxEK1122.A_0027_ER2328_0002_0019.Channel_8.Output <-> Channel 8/Output
//     PlcTask Inputs/GVL_iXlinker.EtherCAT_Master_ERxxxx.Beckhoff_ER2xxx.Beckhoff_ER2xxxEK1122.A_0027_ER2328_0002_0019.WcState.WcState <-> WcState/WcState
//     PlcTask Inputs/GVL_iXlinker.EtherCAT_Master_ERxxxx.Beckhoff_ER2xxx.Beckhoff_ER2xxxEK1122.A_0027_ER2328_0002_0019.WcState.InputToggle <-> WcState/InputToggle
//     PlcTask Inputs/GVL_iXlinker.EtherCAT_Master_ERxxxx.Beckhoff_ER2xxx.Beckhoff_ER2xxxEK1122.A_0027_ER2328_0002_0019.InfoData.State <-> InfoData/State
//   PLC/PLC Instance <-> EtherCAT Master ERxxxx/Beckhoff ER2xxx/Beckhoff ER2xxxEK1122/A_0028(ER2338-0001-0022)
//     PlcTask Inputs/GVL_iXlinker.EtherCAT_Master_ERxxxx.Beckhoff_ER2xxx.Beckhoff_ER2xxxEK1122.A_0028_ER2338_0001_0022.Channel_1.Input <-> Channel 1/Input
//     PlcTask Inputs/GVL_iXlinker.EtherCAT_Master_ERxxxx.Beckhoff_ER2xxx.Beckhoff_ER2xxxEK1122.A_0028_ER2338_0001_0022.Channel_2.Input <-> Channel 2/Input
//     PlcTask Inputs/GVL_iXlinker.EtherCAT_Master_ERxxxx.Beckhoff_ER2xxx.Beckhoff_ER2xxxEK1122.A_0028_ER2338_0001_0022.Channel_3.Input <-> Channel 3/Input
//     PlcTask Inputs/GVL_iXlinker.EtherCAT_Master_ERxxxx.Beckhoff_ER2xxx.Beckhoff_ER2xxxEK1122.A_0028_ER2338_0001_0022.Channel_4.Input <-> Channel 4/Input
//     PlcTask Inputs/GVL_iXlinker.EtherCAT_Master_ERxxxx.Beckhoff_ER2xxx.Beckhoff_ER2xxxEK1122.A_0028_ER2338_0001_0022.Channel_5.Input <-> Channel 5/Input
//     PlcTask Inputs/GVL_iXlinker.EtherCAT_Master_ERxxxx.Beckhoff_ER2xxx.Beckhoff_ER2xxxEK1122.A_0028_ER2338_0001_0022.Channel_6.Input <-> Channel 6/Input
//     PlcTask Inputs/GVL_iXlinker.EtherCAT_Master_ERxxxx.Beckhoff_ER2xxx.Beckhoff_ER2xxxEK1122.A_0028_ER2338_0001_0022.Channel_7.Input <-> Channel 7/Input
//     PlcTask Inputs/GVL_iXlinker.EtherCAT_Master_ERxxxx.Beckhoff_ER2xxx.Beckhoff_ER2xxxEK1122.A_0028_ER2338_0001_0022.Channel_8.Input <-> Channel 8/Input
//     PlcTask Outputs/GVL_iXlinker.EtherCAT_Master_ERxxxx.Beckhoff_ER2xxx.Beckhoff_ER2xxxEK1122.A_0028_ER2338_0001_0022.Channel_9.Output <-> Channel 9/Output
//     PlcTask Outputs/GVL_iXlinker.EtherCAT_Master_ERxxxx.Beckhoff_ER2xxx.Beckhoff_ER2xxxEK1122.A_0028_ER2338_0001_0022.Channel_10.Output <-> Channel 10/Output
//     PlcTask Outputs/GVL_iXlinker.EtherCAT_Master_ERxxxx.Beckhoff_ER2xxx.Beckhoff_ER2xxxEK1122.A_0028_ER2338_0001_0022.Channel_11.Output <-> Channel 11/Output
//     PlcTask Outputs/GVL_iXlinker.EtherCAT_Master_ERxxxx.Beckhoff_ER2xxx.Beckhoff_ER2xxxEK1122.A_0028_ER2338_0001_0022.Channel_12.Output <-> Channel 12/Output
//     PlcTask Outputs/GVL_iXlinker.EtherCAT_Master_ERxxxx.Beckhoff_ER2xxx.Beckhoff_ER2xxxEK1122.A_0028_ER2338_0001_0022.Channel_13.Output <-> Channel 13/Output
//     PlcTask Outputs/GVL_iXlinker.EtherCAT_Master_ERxxxx.Beckhoff_ER2xxx.Beckhoff_ER2xxxEK1122.A_0028_ER2338_0001_0022.Channel_14.Output <-> Channel 14/Output
//     PlcTask Outputs/GVL_iXlinker.EtherCAT_Master_ERxxxx.Beckhoff_ER2xxx.Beckhoff_ER2xxxEK1122.A_0028_ER2338_0001_0022.Channel_15.Output <-> Channel 15/Output
//     PlcTask Outputs/GVL_iXlinker.EtherCAT_Master_ERxxxx.Beckhoff_ER2xxx.Beckhoff_ER2xxxEK1122.A_0028_ER2338_0001_0022.Channel_16.Output <-> Channel 16/Output
//     PlcTask Inputs/GVL_iXlinker.EtherCAT_Master_ERxxxx.Beckhoff_ER2xxx.Beckhoff_ER2xxxEK1122.A_0028_ER2338_0001_0022.WcState.WcState <-> WcState/WcState
//     PlcTask Inputs/GVL_iXlinker.EtherCAT_Master_ERxxxx.Beckhoff_ER2xxx.Beckhoff_ER2xxxEK1122.A_0028_ER2338_0001_0022.WcState.InputToggle <-> WcState/InputToggle
//     PlcTask Inputs/GVL_iXlinker.EtherCAT_Master_ERxxxx.Beckhoff_ER2xxx.Beckhoff_ER2xxxEK1122.A_0028_ER2338_0001_0022.InfoData.State <-> InfoData/State
//   PLC/PLC Instance <-> EtherCAT Master ERxxxx/Beckhoff ER2xxx/Beckhoff ER2xxxEK1122/A_0029(ER2338-0001-0023)
//     PlcTask Inputs/GVL_iXlinker.EtherCAT_Master_ERxxxx.Beckhoff_ER2xxx.Beckhoff_ER2xxxEK1122.A_0029_ER2338_0001_0023.Channel_1.Input <-> Channel 1/Input
//     PlcTask Inputs/GVL_iXlinker.EtherCAT_Master_ERxxxx.Beckhoff_ER2xxx.Beckhoff_ER2xxxEK1122.A_0029_ER2338_0001_0023.Channel_2.Input <-> Channel 2/Input
//     PlcTask Inputs/GVL_iXlinker.EtherCAT_Master_ERxxxx.Beckhoff_ER2xxx.Beckhoff_ER2xxxEK1122.A_0029_ER2338_0001_0023.Channel_3.Input <-> Channel 3/Input
//     PlcTask Inputs/GVL_iXlinker.EtherCAT_Master_ERxxxx.Beckhoff_ER2xxx.Beckhoff_ER2xxxEK1122.A_0029_ER2338_0001_0023.Channel_4.Input <-> Channel 4/Input
//     PlcTask Inputs/GVL_iXlinker.EtherCAT_Master_ERxxxx.Beckhoff_ER2xxx.Beckhoff_ER2xxxEK1122.A_0029_ER2338_0001_0023.Channel_5.Input <-> Channel 5/Input
//     PlcTask Inputs/GVL_iXlinker.EtherCAT_Master_ERxxxx.Beckhoff_ER2xxx.Beckhoff_ER2xxxEK1122.A_0029_ER2338_0001_0023.Channel_6.Input <-> Channel 6/Input
//     PlcTask Inputs/GVL_iXlinker.EtherCAT_Master_ERxxxx.Beckhoff_ER2xxx.Beckhoff_ER2xxxEK1122.A_0029_ER2338_0001_0023.Channel_7.Input <-> Channel 7/Input
//     PlcTask Inputs/GVL_iXlinker.EtherCAT_Master_ERxxxx.Beckhoff_ER2xxx.Beckhoff_ER2xxxEK1122.A_0029_ER2338_0001_0023.Channel_8.Input <-> Channel 8/Input
//     PlcTask Outputs/GVL_iXlinker.EtherCAT_Master_ERxxxx.Beckhoff_ER2xxx.Beckhoff_ER2xxxEK1122.A_0029_ER2338_0001_0023.Channel_9.Output <-> Channel 9/Output
//     PlcTask Outputs/GVL_iXlinker.EtherCAT_Master_ERxxxx.Beckhoff_ER2xxx.Beckhoff_ER2xxxEK1122.A_0029_ER2338_0001_0023.Channel_10.Output <-> Channel 10/Output
//     PlcTask Outputs/GVL_iXlinker.EtherCAT_Master_ERxxxx.Beckhoff_ER2xxx.Beckhoff_ER2xxxEK1122.A_0029_ER2338_0001_0023.Channel_11.Output <-> Channel 11/Output
//     PlcTask Outputs/GVL_iXlinker.EtherCAT_Master_ERxxxx.Beckhoff_ER2xxx.Beckhoff_ER2xxxEK1122.A_0029_ER2338_0001_0023.Channel_12.Output <-> Channel 12/Output
//     PlcTask Outputs/GVL_iXlinker.EtherCAT_Master_ERxxxx.Beckhoff_ER2xxx.Beckhoff_ER2xxxEK1122.A_0029_ER2338_0001_0023.Channel_13.Output <-> Channel 13/Output
//     PlcTask Outputs/GVL_iXlinker.EtherCAT_Master_ERxxxx.Beckhoff_ER2xxx.Beckhoff_ER2xxxEK1122.A_0029_ER2338_0001_0023.Channel_14.Output <-> Channel 14/Output
//     PlcTask Outputs/GVL_iXlinker.EtherCAT_Master_ERxxxx.Beckhoff_ER2xxx.Beckhoff_ER2xxxEK1122.A_0029_ER2338_0001_0023.Channel_15.Output <-> Channel 15/Output
//     PlcTask Outputs/GVL_iXlinker.EtherCAT_Master_ERxxxx.Beckhoff_ER2xxx.Beckhoff_ER2xxxEK1122.A_0029_ER2338_0001_0023.Channel_16.Output <-> Channel 16/Output
//     PlcTask Inputs/GVL_iXlinker.EtherCAT_Master_ERxxxx.Beckhoff_ER2xxx.Beckhoff_ER2xxxEK1122.A_0029_ER2338_0001_0023.WcState.WcState <-> WcState/WcState
//     PlcTask Inputs/GVL_iXlinker.EtherCAT_Master_ERxxxx.Beckhoff_ER2xxx.Beckhoff_ER2xxxEK1122.A_0029_ER2338_0001_0023.WcState.InputToggle <-> WcState/InputToggle
//     PlcTask Inputs/GVL_iXlinker.EtherCAT_Master_ERxxxx.Beckhoff_ER2xxx.Beckhoff_ER2xxxEK1122.A_0029_ER2338_0001_0023.InfoData.State <-> InfoData/State
//   PLC/PLC Instance <-> EtherCAT Master ERxxxx/Beckhoff ER2xxx/Beckhoff ER2xxxEK1122/A_0030(ER2338-0002-0022)
//     PlcTask Inputs/GVL_iXlinker.EtherCAT_Master_ERxxxx.Beckhoff_ER2xxx.Beckhoff_ER2xxxEK1122.A_0030_ER2338_0002_0022.Channel_1.Input <-> Channel 1/Input
//     PlcTask Inputs/GVL_iXlinker.EtherCAT_Master_ERxxxx.Beckhoff_ER2xxx.Beckhoff_ER2xxxEK1122.A_0030_ER2338_0002_0022.Channel_2.Input <-> Channel 2/Input
//     PlcTask Inputs/GVL_iXlinker.EtherCAT_Master_ERxxxx.Beckhoff_ER2xxx.Beckhoff_ER2xxxEK1122.A_0030_ER2338_0002_0022.Channel_3.Input <-> Channel 3/Input
//     PlcTask Inputs/GVL_iXlinker.EtherCAT_Master_ERxxxx.Beckhoff_ER2xxx.Beckhoff_ER2xxxEK1122.A_0030_ER2338_0002_0022.Channel_4.Input <-> Channel 4/Input
//     PlcTask Inputs/GVL_iXlinker.EtherCAT_Master_ERxxxx.Beckhoff_ER2xxx.Beckhoff_ER2xxxEK1122.A_0030_ER2338_0002_0022.Channel_5.Input <-> Channel 5/Input
//     PlcTask Inputs/GVL_iXlinker.EtherCAT_Master_ERxxxx.Beckhoff_ER2xxx.Beckhoff_ER2xxxEK1122.A_0030_ER2338_0002_0022.Channel_6.Input <-> Channel 6/Input
//     PlcTask Inputs/GVL_iXlinker.EtherCAT_Master_ERxxxx.Beckhoff_ER2xxx.Beckhoff_ER2xxxEK1122.A_0030_ER2338_0002_0022.Channel_7.Input <-> Channel 7/Input
//     PlcTask Inputs/GVL_iXlinker.EtherCAT_Master_ERxxxx.Beckhoff_ER2xxx.Beckhoff_ER2xxxEK1122.A_0030_ER2338_0002_0022.Channel_8.Input <-> Channel 8/Input
//     PlcTask Outputs/GVL_iXlinker.EtherCAT_Master_ERxxxx.Beckhoff_ER2xxx.Beckhoff_ER2xxxEK1122.A_0030_ER2338_0002_0022.Channel_9.Output <-> Channel 9/Output
//     PlcTask Outputs/GVL_iXlinker.EtherCAT_Master_ERxxxx.Beckhoff_ER2xxx.Beckhoff_ER2xxxEK1122.A_0030_ER2338_0002_0022.Channel_10.Output <-> Channel 10/Output
//     PlcTask Outputs/GVL_iXlinker.EtherCAT_Master_ERxxxx.Beckhoff_ER2xxx.Beckhoff_ER2xxxEK1122.A_0030_ER2338_0002_0022.Channel_11.Output <-> Channel 11/Output
//     PlcTask Outputs/GVL_iXlinker.EtherCAT_Master_ERxxxx.Beckhoff_ER2xxx.Beckhoff_ER2xxxEK1122.A_0030_ER2338_0002_0022.Channel_12.Output <-> Channel 12/Output
//     PlcTask Outputs/GVL_iXlinker.EtherCAT_Master_ERxxxx.Beckhoff_ER2xxx.Beckhoff_ER2xxxEK1122.A_0030_ER2338_0002_0022.Channel_13.Output <-> Channel 13/Output
//     PlcTask Outputs/GVL_iXlinker.EtherCAT_Master_ERxxxx.Beckhoff_ER2xxx.Beckhoff_ER2xxxEK1122.A_0030_ER2338_0002_0022.Channel_14.Output <-> Channel 14/Output
//     PlcTask Outputs/GVL_iXlinker.EtherCAT_Master_ERxxxx.Beckhoff_ER2xxx.Beckhoff_ER2xxxEK1122.A_0030_ER2338_0002_0022.Channel_15.Output <-> Channel 15/Output
//     PlcTask Outputs/GVL_iXlinker.EtherCAT_Master_ERxxxx.Beckhoff_ER2xxx.Beckhoff_ER2xxxEK1122.A_0030_ER2338_0002_0022.Channel_16.Output <-> Channel 16/Output
//     PlcTask Inputs/GVL_iXlinker.EtherCAT_Master_ERxxxx.Beckhoff_ER2xxx.Beckhoff_ER2xxxEK1122.A_0030_ER2338_0002_0022.WcState.WcState <-> WcState/WcState
//     PlcTask Inputs/GVL_iXlinker.EtherCAT_Master_ERxxxx.Beckhoff_ER2xxx.Beckhoff_ER2xxxEK1122.A_0030_ER2338_0002_0022.WcState.InputToggle <-> WcState/InputToggle
//     PlcTask Inputs/GVL_iXlinker.EtherCAT_Master_ERxxxx.Beckhoff_ER2xxx.Beckhoff_ER2xxxEK1122.A_0030_ER2338_0002_0022.InfoData.State <-> InfoData/State
//   PLC/PLC Instance <-> EtherCAT Master ERxxxx/Beckhoff ER2xxx/Beckhoff ER2xxxEK1122/A_0031(ER2338-0002-0023)
//     PlcTask Inputs/GVL_iXlinker.EtherCAT_Master_ERxxxx.Beckhoff_ER2xxx.Beckhoff_ER2xxxEK1122.A_0031_ER2338_0002_0023.Channel_1.Input <-> Channel 1/Input
//     PlcTask Inputs/GVL_iXlinker.EtherCAT_Master_ERxxxx.Beckhoff_ER2xxx.Beckhoff_ER2xxxEK1122.A_0031_ER2338_0002_0023.Channel_2.Input <-> Channel 2/Input
//     PlcTask Inputs/GVL_iXlinker.EtherCAT_Master_ERxxxx.Beckhoff_ER2xxx.Beckhoff_ER2xxxEK1122.A_0031_ER2338_0002_0023.Channel_3.Input <-> Channel 3/Input
//     PlcTask Inputs/GVL_iXlinker.EtherCAT_Master_ERxxxx.Beckhoff_ER2xxx.Beckhoff_ER2xxxEK1122.A_0031_ER2338_0002_0023.Channel_4.Input <-> Channel 4/Input
//     PlcTask Inputs/GVL_iXlinker.EtherCAT_Master_ERxxxx.Beckhoff_ER2xxx.Beckhoff_ER2xxxEK1122.A_0031_ER2338_0002_0023.Channel_5.Input <-> Channel 5/Input
//     PlcTask Inputs/GVL_iXlinker.EtherCAT_Master_ERxxxx.Beckhoff_ER2xxx.Beckhoff_ER2xxxEK1122.A_0031_ER2338_0002_0023.Channel_6.Input <-> Channel 6/Input
//     PlcTask Inputs/GVL_iXlinker.EtherCAT_Master_ERxxxx.Beckhoff_ER2xxx.Beckhoff_ER2xxxEK1122.A_0031_ER2338_0002_0023.Channel_7.Input <-> Channel 7/Input
//     PlcTask Inputs/GVL_iXlinker.EtherCAT_Master_ERxxxx.Beckhoff_ER2xxx.Beckhoff_ER2xxxEK1122.A_0031_ER2338_0002_0023.Channel_8.Input <-> Channel 8/Input
//     PlcTask Outputs/GVL_iXlinker.EtherCAT_Master_ERxxxx.Beckhoff_ER2xxx.Beckhoff_ER2xxxEK1122.A_0031_ER2338_0002_0023.Channel_9.Output <-> Channel 9/Output
//     PlcTask Outputs/GVL_iXlinker.EtherCAT_Master_ERxxxx.Beckhoff_ER2xxx.Beckhoff_ER2xxxEK1122.A_0031_ER2338_0002_0023.Channel_10.Output <-> Channel 10/Output
//     PlcTask Outputs/GVL_iXlinker.EtherCAT_Master_ERxxxx.Beckhoff_ER2xxx.Beckhoff_ER2xxxEK1122.A_0031_ER2338_0002_0023.Channel_11.Output <-> Channel 11/Output
//     PlcTask Outputs/GVL_iXlinker.EtherCAT_Master_ERxxxx.Beckhoff_ER2xxx.Beckhoff_ER2xxxEK1122.A_0031_ER2338_0002_0023.Channel_12.Output <-> Channel 12/Output
//     PlcTask Outputs/GVL_iXlinker.EtherCAT_Master_ERxxxx.Beckhoff_ER2xxx.Beckhoff_ER2xxxEK1122.A_0031_ER2338_0002_0023.Channel_13.Output <-> Channel 13/Output
//     PlcTask Outputs/GVL_iXlinker.EtherCAT_Master_ERxxxx.Beckhoff_ER2xxx.Beckhoff_ER2xxxEK1122.A_0031_ER2338_0002_0023.Channel_14.Output <-> Channel 14/Output
//     PlcTask Outputs/GVL_iXlinker.EtherCAT_Master_ERxxxx.Beckhoff_ER2xxx.Beckhoff_ER2xxxEK1122.A_0031_ER2338_0002_0023.Channel_15.Output <-> Channel 15/Output
//     PlcTask Outputs/GVL_iXlinker.EtherCAT_Master_ERxxxx.Beckhoff_ER2xxx.Beckhoff_ER2xxxEK1122.A_0031_ER2338_0002_0023.Channel_16.Output <-> Channel 16/Output
//     PlcTask Inputs/GVL_iXlinker.EtherCAT_Master_ERxxxx.Beckhoff_ER2xxx.Beckhoff_ER2xxxEK1122.A_0031_ER2338_0002_0023.WcState.WcState <-> WcState/WcState
//     PlcTask Inputs/GVL_iXlinker.EtherCAT_Master_ERxxxx.Beckhoff_ER2xxx.Beckhoff_ER2xxxEK1122.A_0031_ER2338_0002_0023.WcState.InputToggle <-> WcState/InputToggle
//     PlcTask Inputs/GVL_iXlinker.EtherCAT_Master_ERxxxx.Beckhoff_ER2xxx.Beckhoff_ER2xxxEK1122.A_0031_ER2338_0002_0023.InfoData.State <-> InfoData/State
//   PLC/PLC Instance <-> EtherCAT Master ERxxxx/Beckhoff ER2xxx/Beckhoff ER2xxxEK1122/A_0032(ER2338-1001-0017)
//     PlcTask Inputs/GVL_iXlinker.EtherCAT_Master_ERxxxx.Beckhoff_ER2xxx.Beckhoff_ER2xxxEK1122.A_0032_ER2338_1001_0017.Channel_1.Input <-> Channel 1/Input
//     PlcTask Inputs/GVL_iXlinker.EtherCAT_Master_ERxxxx.Beckhoff_ER2xxx.Beckhoff_ER2xxxEK1122.A_0032_ER2338_1001_0017.Channel_2.Input <-> Channel 2/Input
//     PlcTask Inputs/GVL_iXlinker.EtherCAT_Master_ERxxxx.Beckhoff_ER2xxx.Beckhoff_ER2xxxEK1122.A_0032_ER2338_1001_0017.Channel_3.Input <-> Channel 3/Input
//     PlcTask Inputs/GVL_iXlinker.EtherCAT_Master_ERxxxx.Beckhoff_ER2xxx.Beckhoff_ER2xxxEK1122.A_0032_ER2338_1001_0017.Channel_4.Input <-> Channel 4/Input
//     PlcTask Inputs/GVL_iXlinker.EtherCAT_Master_ERxxxx.Beckhoff_ER2xxx.Beckhoff_ER2xxxEK1122.A_0032_ER2338_1001_0017.Channel_5.Input <-> Channel 5/Input
//     PlcTask Inputs/GVL_iXlinker.EtherCAT_Master_ERxxxx.Beckhoff_ER2xxx.Beckhoff_ER2xxxEK1122.A_0032_ER2338_1001_0017.Channel_6.Input <-> Channel 6/Input
//     PlcTask Inputs/GVL_iXlinker.EtherCAT_Master_ERxxxx.Beckhoff_ER2xxx.Beckhoff_ER2xxxEK1122.A_0032_ER2338_1001_0017.Channel_7.Input <-> Channel 7/Input
//     PlcTask Inputs/GVL_iXlinker.EtherCAT_Master_ERxxxx.Beckhoff_ER2xxx.Beckhoff_ER2xxxEK1122.A_0032_ER2338_1001_0017.Channel_8.Input <-> Channel 8/Input
//     PlcTask Outputs/GVL_iXlinker.EtherCAT_Master_ERxxxx.Beckhoff_ER2xxx.Beckhoff_ER2xxxEK1122.A_0032_ER2338_1001_0017.Channel_9.Output <-> Channel 9/Output
//     PlcTask Outputs/GVL_iXlinker.EtherCAT_Master_ERxxxx.Beckhoff_ER2xxx.Beckhoff_ER2xxxEK1122.A_0032_ER2338_1001_0017.Channel_10.Output <-> Channel 10/Output
//     PlcTask Outputs/GVL_iXlinker.EtherCAT_Master_ERxxxx.Beckhoff_ER2xxx.Beckhoff_ER2xxxEK1122.A_0032_ER2338_1001_0017.Channel_11.Output <-> Channel 11/Output
//     PlcTask Outputs/GVL_iXlinker.EtherCAT_Master_ERxxxx.Beckhoff_ER2xxx.Beckhoff_ER2xxxEK1122.A_0032_ER2338_1001_0017.Channel_12.Output <-> Channel 12/Output
//     PlcTask Outputs/GVL_iXlinker.EtherCAT_Master_ERxxxx.Beckhoff_ER2xxx.Beckhoff_ER2xxxEK1122.A_0032_ER2338_1001_0017.Channel_13.Output <-> Channel 13/Output
//     PlcTask Outputs/GVL_iXlinker.EtherCAT_Master_ERxxxx.Beckhoff_ER2xxx.Beckhoff_ER2xxxEK1122.A_0032_ER2338_1001_0017.Channel_14.Output <-> Channel 14/Output
//     PlcTask Outputs/GVL_iXlinker.EtherCAT_Master_ERxxxx.Beckhoff_ER2xxx.Beckhoff_ER2xxxEK1122.A_0032_ER2338_1001_0017.Channel_15.Output <-> Channel 15/Output
//     PlcTask Outputs/GVL_iXlinker.EtherCAT_Master_ERxxxx.Beckhoff_ER2xxx.Beckhoff_ER2xxxEK1122.A_0032_ER2338_1001_0017.Channel_16.Output <-> Channel 16/Output
//     PlcTask Inputs/GVL_iXlinker.EtherCAT_Master_ERxxxx.Beckhoff_ER2xxx.Beckhoff_ER2xxxEK1122.A_0032_ER2338_1001_0017.WcState.WcState <-> WcState/WcState
//     PlcTask Inputs/GVL_iXlinker.EtherCAT_Master_ERxxxx.Beckhoff_ER2xxx.Beckhoff_ER2xxxEK1122.A_0032_ER2338_1001_0017.WcState.InputToggle <-> WcState/InputToggle
//     PlcTask Inputs/GVL_iXlinker.EtherCAT_Master_ERxxxx.Beckhoff_ER2xxx.Beckhoff_ER2xxxEK1122.A_0032_ER2338_1001_0017.InfoData.State <-> InfoData/State
//   PLC/PLC Instance <-> EtherCAT Master ERxxxx/Beckhoff ER2xxx/Beckhoff ER2xxxEK1122/A_0033(ER2338-1001-0018)
//     PlcTask Inputs/GVL_iXlinker.EtherCAT_Master_ERxxxx.Beckhoff_ER2xxx.Beckhoff_ER2xxxEK1122.A_0033_ER2338_1001_0018.Channel_1.Input <-> Channel 1/Input
//     PlcTask Inputs/GVL_iXlinker.EtherCAT_Master_ERxxxx.Beckhoff_ER2xxx.Beckhoff_ER2xxxEK1122.A_0033_ER2338_1001_0018.Channel_2.Input <-> Channel 2/Input
//     PlcTask Inputs/GVL_iXlinker.EtherCAT_Master_ERxxxx.Beckhoff_ER2xxx.Beckhoff_ER2xxxEK1122.A_0033_ER2338_1001_0018.Channel_3.Input <-> Channel 3/Input
//     PlcTask Inputs/GVL_iXlinker.EtherCAT_Master_ERxxxx.Beckhoff_ER2xxx.Beckhoff_ER2xxxEK1122.A_0033_ER2338_1001_0018.Channel_4.Input <-> Channel 4/Input
//     PlcTask Inputs/GVL_iXlinker.EtherCAT_Master_ERxxxx.Beckhoff_ER2xxx.Beckhoff_ER2xxxEK1122.A_0033_ER2338_1001_0018.Channel_5.Input <-> Channel 5/Input
//     PlcTask Inputs/GVL_iXlinker.EtherCAT_Master_ERxxxx.Beckhoff_ER2xxx.Beckhoff_ER2xxxEK1122.A_0033_ER2338_1001_0018.Channel_6.Input <-> Channel 6/Input
//     PlcTask Inputs/GVL_iXlinker.EtherCAT_Master_ERxxxx.Beckhoff_ER2xxx.Beckhoff_ER2xxxEK1122.A_0033_ER2338_1001_0018.Channel_7.Input <-> Channel 7/Input
//     PlcTask Inputs/GVL_iXlinker.EtherCAT_Master_ERxxxx.Beckhoff_ER2xxx.Beckhoff_ER2xxxEK1122.A_0033_ER2338_1001_0018.Channel_8.Input <-> Channel 8/Input
//     PlcTask Outputs/GVL_iXlinker.EtherCAT_Master_ERxxxx.Beckhoff_ER2xxx.Beckhoff_ER2xxxEK1122.A_0033_ER2338_1001_0018.Channel_9.Output <-> Channel 9/Output
//     PlcTask Outputs/GVL_iXlinker.EtherCAT_Master_ERxxxx.Beckhoff_ER2xxx.Beckhoff_ER2xxxEK1122.A_0033_ER2338_1001_0018.Channel_10.Output <-> Channel 10/Output
//     PlcTask Outputs/GVL_iXlinker.EtherCAT_Master_ERxxxx.Beckhoff_ER2xxx.Beckhoff_ER2xxxEK1122.A_0033_ER2338_1001_0018.Channel_11.Output <-> Channel 11/Output
//     PlcTask Outputs/GVL_iXlinker.EtherCAT_Master_ERxxxx.Beckhoff_ER2xxx.Beckhoff_ER2xxxEK1122.A_0033_ER2338_1001_0018.Channel_12.Output <-> Channel 12/Output
//     PlcTask Outputs/GVL_iXlinker.EtherCAT_Master_ERxxxx.Beckhoff_ER2xxx.Beckhoff_ER2xxxEK1122.A_0033_ER2338_1001_0018.Channel_13.Output <-> Channel 13/Output
//     PlcTask Outputs/GVL_iXlinker.EtherCAT_Master_ERxxxx.Beckhoff_ER2xxx.Beckhoff_ER2xxxEK1122.A_0033_ER2338_1001_0018.Channel_14.Output <-> Channel 14/Output
//     PlcTask Outputs/GVL_iXlinker.EtherCAT_Master_ERxxxx.Beckhoff_ER2xxx.Beckhoff_ER2xxxEK1122.A_0033_ER2338_1001_0018.Channel_15.Output <-> Channel 15/Output
//     PlcTask Outputs/GVL_iXlinker.EtherCAT_Master_ERxxxx.Beckhoff_ER2xxx.Beckhoff_ER2xxxEK1122.A_0033_ER2338_1001_0018.Channel_16.Output <-> Channel 16/Output
//     PlcTask Inputs/GVL_iXlinker.EtherCAT_Master_ERxxxx.Beckhoff_ER2xxx.Beckhoff_ER2xxxEK1122.A_0033_ER2338_1001_0018.WcState.WcState <-> WcState/WcState
//     PlcTask Inputs/GVL_iXlinker.EtherCAT_Master_ERxxxx.Beckhoff_ER2xxx.Beckhoff_ER2xxxEK1122.A_0033_ER2338_1001_0018.WcState.InputToggle <-> WcState/InputToggle
//     PlcTask Inputs/GVL_iXlinker.EtherCAT_Master_ERxxxx.Beckhoff_ER2xxx.Beckhoff_ER2xxxEK1122.A_0033_ER2338_1001_0018.InfoData.State <-> InfoData/State
//   PLC/PLC Instance <-> EtherCAT Master ERxxxx/Beckhoff ER2xxx/Beckhoff ER2xxxEK1122/A_0034(ER2338-1002-0017)
//     PlcTask Inputs/GVL_iXlinker.EtherCAT_Master_ERxxxx.Beckhoff_ER2xxx.Beckhoff_ER2xxxEK1122.A_0034_ER2338_1002_0017.Channel_1.Input <-> Channel 1/Input
//     PlcTask Inputs/GVL_iXlinker.EtherCAT_Master_ERxxxx.Beckhoff_ER2xxx.Beckhoff_ER2xxxEK1122.A_0034_ER2338_1002_0017.Channel_2.Input <-> Channel 2/Input
//     PlcTask Inputs/GVL_iXlinker.EtherCAT_Master_ERxxxx.Beckhoff_ER2xxx.Beckhoff_ER2xxxEK1122.A_0034_ER2338_1002_0017.Channel_3.Input <-> Channel 3/Input
//     PlcTask Inputs/GVL_iXlinker.EtherCAT_Master_ERxxxx.Beckhoff_ER2xxx.Beckhoff_ER2xxxEK1122.A_0034_ER2338_1002_0017.Channel_4.Input <-> Channel 4/Input
//     PlcTask Inputs/GVL_iXlinker.EtherCAT_Master_ERxxxx.Beckhoff_ER2xxx.Beckhoff_ER2xxxEK1122.A_0034_ER2338_1002_0017.Channel_5.Input <-> Channel 5/Input
//     PlcTask Inputs/GVL_iXlinker.EtherCAT_Master_ERxxxx.Beckhoff_ER2xxx.Beckhoff_ER2xxxEK1122.A_0034_ER2338_1002_0017.Channel_6.Input <-> Channel 6/Input
//     PlcTask Inputs/GVL_iXlinker.EtherCAT_Master_ERxxxx.Beckhoff_ER2xxx.Beckhoff_ER2xxxEK1122.A_0034_ER2338_1002_0017.Channel_7.Input <-> Channel 7/Input
//     PlcTask Inputs/GVL_iXlinker.EtherCAT_Master_ERxxxx.Beckhoff_ER2xxx.Beckhoff_ER2xxxEK1122.A_0034_ER2338_1002_0017.Channel_8.Input <-> Channel 8/Input
//     PlcTask Outputs/GVL_iXlinker.EtherCAT_Master_ERxxxx.Beckhoff_ER2xxx.Beckhoff_ER2xxxEK1122.A_0034_ER2338_1002_0017.Channel_9.Output <-> Channel 9/Output
//     PlcTask Outputs/GVL_iXlinker.EtherCAT_Master_ERxxxx.Beckhoff_ER2xxx.Beckhoff_ER2xxxEK1122.A_0034_ER2338_1002_0017.Channel_10.Output <-> Channel 10/Output
//     PlcTask Outputs/GVL_iXlinker.EtherCAT_Master_ERxxxx.Beckhoff_ER2xxx.Beckhoff_ER2xxxEK1122.A_0034_ER2338_1002_0017.Channel_11.Output <-> Channel 11/Output
//     PlcTask Outputs/GVL_iXlinker.EtherCAT_Master_ERxxxx.Beckhoff_ER2xxx.Beckhoff_ER2xxxEK1122.A_0034_ER2338_1002_0017.Channel_12.Output <-> Channel 12/Output
//     PlcTask Outputs/GVL_iXlinker.EtherCAT_Master_ERxxxx.Beckhoff_ER2xxx.Beckhoff_ER2xxxEK1122.A_0034_ER2338_1002_0017.Channel_13.Output <-> Channel 13/Output
//     PlcTask Outputs/GVL_iXlinker.EtherCAT_Master_ERxxxx.Beckhoff_ER2xxx.Beckhoff_ER2xxxEK1122.A_0034_ER2338_1002_0017.Channel_14.Output <-> Channel 14/Output
//     PlcTask Outputs/GVL_iXlinker.EtherCAT_Master_ERxxxx.Beckhoff_ER2xxx.Beckhoff_ER2xxxEK1122.A_0034_ER2338_1002_0017.Channel_15.Output <-> Channel 15/Output
//     PlcTask Outputs/GVL_iXlinker.EtherCAT_Master_ERxxxx.Beckhoff_ER2xxx.Beckhoff_ER2xxxEK1122.A_0034_ER2338_1002_0017.Channel_16.Output <-> Channel 16/Output
//     PlcTask Inputs/GVL_iXlinker.EtherCAT_Master_ERxxxx.Beckhoff_ER2xxx.Beckhoff_ER2xxxEK1122.A_0034_ER2338_1002_0017.WcState.WcState <-> WcState/WcState
//     PlcTask Inputs/GVL_iXlinker.EtherCAT_Master_ERxxxx.Beckhoff_ER2xxx.Beckhoff_ER2xxxEK1122.A_0034_ER2338_1002_0017.WcState.InputToggle <-> WcState/InputToggle
//     PlcTask Inputs/GVL_iXlinker.EtherCAT_Master_ERxxxx.Beckhoff_ER2xxx.Beckhoff_ER2xxxEK1122.A_0034_ER2338_1002_0017.InfoData.State <-> InfoData/State
//   PLC/PLC Instance <-> EtherCAT Master ERxxxx/Beckhoff ER2xxx/Beckhoff ER2xxxEK1122/A_0035(ER2338-1002-0018)
//     PlcTask Inputs/GVL_iXlinker.EtherCAT_Master_ERxxxx.Beckhoff_ER2xxx.Beckhoff_ER2xxxEK1122.A_0035_ER2338_1002_0018.Channel_1.Input <-> Channel 1/Input
//     PlcTask Inputs/GVL_iXlinker.EtherCAT_Master_ERxxxx.Beckhoff_ER2xxx.Beckhoff_ER2xxxEK1122.A_0035_ER2338_1002_0018.Channel_2.Input <-> Channel 2/Input
//     PlcTask Inputs/GVL_iXlinker.EtherCAT_Master_ERxxxx.Beckhoff_ER2xxx.Beckhoff_ER2xxxEK1122.A_0035_ER2338_1002_0018.Channel_3.Input <-> Channel 3/Input
//     PlcTask Inputs/GVL_iXlinker.EtherCAT_Master_ERxxxx.Beckhoff_ER2xxx.Beckhoff_ER2xxxEK1122.A_0035_ER2338_1002_0018.Channel_4.Input <-> Channel 4/Input
//     PlcTask Inputs/GVL_iXlinker.EtherCAT_Master_ERxxxx.Beckhoff_ER2xxx.Beckhoff_ER2xxxEK1122.A_0035_ER2338_1002_0018.Channel_5.Input <-> Channel 5/Input
//     PlcTask Inputs/GVL_iXlinker.EtherCAT_Master_ERxxxx.Beckhoff_ER2xxx.Beckhoff_ER2xxxEK1122.A_0035_ER2338_1002_0018.Channel_6.Input <-> Channel 6/Input
//     PlcTask Inputs/GVL_iXlinker.EtherCAT_Master_ERxxxx.Beckhoff_ER2xxx.Beckhoff_ER2xxxEK1122.A_0035_ER2338_1002_0018.Channel_7.Input <-> Channel 7/Input
//     PlcTask Inputs/GVL_iXlinker.EtherCAT_Master_ERxxxx.Beckhoff_ER2xxx.Beckhoff_ER2xxxEK1122.A_0035_ER2338_1002_0018.Channel_8.Input <-> Channel 8/Input
//     PlcTask Outputs/GVL_iXlinker.EtherCAT_Master_ERxxxx.Beckhoff_ER2xxx.Beckhoff_ER2xxxEK1122.A_0035_ER2338_1002_0018.Channel_9.Output <-> Channel 9/Output
//     PlcTask Outputs/GVL_iXlinker.EtherCAT_Master_ERxxxx.Beckhoff_ER2xxx.Beckhoff_ER2xxxEK1122.A_0035_ER2338_1002_0018.Channel_10.Output <-> Channel 10/Output
//     PlcTask Outputs/GVL_iXlinker.EtherCAT_Master_ERxxxx.Beckhoff_ER2xxx.Beckhoff_ER2xxxEK1122.A_0035_ER2338_1002_0018.Channel_11.Output <-> Channel 11/Output
//     PlcTask Outputs/GVL_iXlinker.EtherCAT_Master_ERxxxx.Beckhoff_ER2xxx.Beckhoff_ER2xxxEK1122.A_0035_ER2338_1002_0018.Channel_12.Output <-> Channel 12/Output
//     PlcTask Outputs/GVL_iXlinker.EtherCAT_Master_ERxxxx.Beckhoff_ER2xxx.Beckhoff_ER2xxxEK1122.A_0035_ER2338_1002_0018.Channel_13.Output <-> Channel 13/Output
//     PlcTask Outputs/GVL_iXlinker.EtherCAT_Master_ERxxxx.Beckhoff_ER2xxx.Beckhoff_ER2xxxEK1122.A_0035_ER2338_1002_0018.Channel_14.Output <-> Channel 14/Output
//     PlcTask Outputs/GVL_iXlinker.EtherCAT_Master_ERxxxx.Beckhoff_ER2xxx.Beckhoff_ER2xxxEK1122.A_0035_ER2338_1002_0018.Channel_15.Output <-> Channel 15/Output
//     PlcTask Outputs/GVL_iXlinker.EtherCAT_Master_ERxxxx.Beckhoff_ER2xxx.Beckhoff_ER2xxxEK1122.A_0035_ER2338_1002_0018.Channel_16.Output <-> Channel 16/Output
//     PlcTask Inputs/GVL_iXlinker.EtherCAT_Master_ERxxxx.Beckhoff_ER2xxx.Beckhoff_ER2xxxEK1122.A_0035_ER2338_1002_0018.WcState.WcState <-> WcState/WcState
//     PlcTask Inputs/GVL_iXlinker.EtherCAT_Master_ERxxxx.Beckhoff_ER2xxx.Beckhoff_ER2xxxEK1122.A_0035_ER2338_1002_0018.WcState.InputToggle <-> WcState/InputToggle
//     PlcTask Inputs/GVL_iXlinker.EtherCAT_Master_ERxxxx.Beckhoff_ER2xxx.Beckhoff_ER2xxxEK1122.A_0035_ER2338_1002_0018.InfoData.State <-> InfoData/State
//   PLC/PLC Instance <-> EtherCAT Master ERxxxx/Beckhoff ER2xxx/Beckhoff ER2xxxEK1122/A_0036(ER2339-0021-0018)
//     PlcTask Inputs/GVL_iXlinker.EtherCAT_Master_ERxxxx.Beckhoff_ER2xxx.Beckhoff_ER2xxxEK1122.A_0036_ER2339_0021_0018.Channel_1.Input <-> Channel 1/Input
//     PlcTask Inputs/GVL_iXlinker.EtherCAT_Master_ERxxxx.Beckhoff_ER2xxx.Beckhoff_ER2xxxEK1122.A_0036_ER2339_0021_0018.Channel_2.Input <-> Channel 2/Input
//     PlcTask Inputs/GVL_iXlinker.EtherCAT_Master_ERxxxx.Beckhoff_ER2xxx.Beckhoff_ER2xxxEK1122.A_0036_ER2339_0021_0018.Channel_3.Input <-> Channel 3/Input
//     PlcTask Inputs/GVL_iXlinker.EtherCAT_Master_ERxxxx.Beckhoff_ER2xxx.Beckhoff_ER2xxxEK1122.A_0036_ER2339_0021_0018.Channel_4.Input <-> Channel 4/Input
//     PlcTask Inputs/GVL_iXlinker.EtherCAT_Master_ERxxxx.Beckhoff_ER2xxx.Beckhoff_ER2xxxEK1122.A_0036_ER2339_0021_0018.Channel_5.Input <-> Channel 5/Input
//     PlcTask Inputs/GVL_iXlinker.EtherCAT_Master_ERxxxx.Beckhoff_ER2xxx.Beckhoff_ER2xxxEK1122.A_0036_ER2339_0021_0018.Channel_6.Input <-> Channel 6/Input
//     PlcTask Inputs/GVL_iXlinker.EtherCAT_Master_ERxxxx.Beckhoff_ER2xxx.Beckhoff_ER2xxxEK1122.A_0036_ER2339_0021_0018.Channel_7.Input <-> Channel 7/Input
//     PlcTask Inputs/GVL_iXlinker.EtherCAT_Master_ERxxxx.Beckhoff_ER2xxx.Beckhoff_ER2xxxEK1122.A_0036_ER2339_0021_0018.Channel_8.Input <-> Channel 8/Input
//     PlcTask Inputs/GVL_iXlinker.EtherCAT_Master_ERxxxx.Beckhoff_ER2xxx.Beckhoff_ER2xxxEK1122.A_0036_ER2339_0021_0018.Channel_9.Input <-> Channel 9/Input
//     PlcTask Inputs/GVL_iXlinker.EtherCAT_Master_ERxxxx.Beckhoff_ER2xxx.Beckhoff_ER2xxxEK1122.A_0036_ER2339_0021_0018.Channel_10.Input <-> Channel 10/Input
//     PlcTask Inputs/GVL_iXlinker.EtherCAT_Master_ERxxxx.Beckhoff_ER2xxx.Beckhoff_ER2xxxEK1122.A_0036_ER2339_0021_0018.Channel_11.Input <-> Channel 11/Input
//     PlcTask Inputs/GVL_iXlinker.EtherCAT_Master_ERxxxx.Beckhoff_ER2xxx.Beckhoff_ER2xxxEK1122.A_0036_ER2339_0021_0018.Channel_12.Input <-> Channel 12/Input
//     PlcTask Inputs/GVL_iXlinker.EtherCAT_Master_ERxxxx.Beckhoff_ER2xxx.Beckhoff_ER2xxxEK1122.A_0036_ER2339_0021_0018.Channel_13.Input <-> Channel 13/Input
//     PlcTask Inputs/GVL_iXlinker.EtherCAT_Master_ERxxxx.Beckhoff_ER2xxx.Beckhoff_ER2xxxEK1122.A_0036_ER2339_0021_0018.Channel_14.Input <-> Channel 14/Input
//     PlcTask Inputs/GVL_iXlinker.EtherCAT_Master_ERxxxx.Beckhoff_ER2xxx.Beckhoff_ER2xxxEK1122.A_0036_ER2339_0021_0018.Channel_15.Input <-> Channel 15/Input
//     PlcTask Inputs/GVL_iXlinker.EtherCAT_Master_ERxxxx.Beckhoff_ER2xxx.Beckhoff_ER2xxxEK1122.A_0036_ER2339_0021_0018.Channel_16.Input <-> Channel 16/Input
//     PlcTask Outputs/GVL_iXlinker.EtherCAT_Master_ERxxxx.Beckhoff_ER2xxx.Beckhoff_ER2xxxEK1122.A_0036_ER2339_0021_0018.Channel_17.Output <-> Channel 17/Output
//     PlcTask Outputs/GVL_iXlinker.EtherCAT_Master_ERxxxx.Beckhoff_ER2xxx.Beckhoff_ER2xxxEK1122.A_0036_ER2339_0021_0018.Channel_18.Output <-> Channel 18/Output
//     PlcTask Outputs/GVL_iXlinker.EtherCAT_Master_ERxxxx.Beckhoff_ER2xxx.Beckhoff_ER2xxxEK1122.A_0036_ER2339_0021_0018.Channel_19.Output <-> Channel 19/Output
//     PlcTask Outputs/GVL_iXlinker.EtherCAT_Master_ERxxxx.Beckhoff_ER2xxx.Beckhoff_ER2xxxEK1122.A_0036_ER2339_0021_0018.Channel_20.Output <-> Channel 20/Output
//     PlcTask Outputs/GVL_iXlinker.EtherCAT_Master_ERxxxx.Beckhoff_ER2xxx.Beckhoff_ER2xxxEK1122.A_0036_ER2339_0021_0018.Channel_21.Output <-> Channel 21/Output
//     PlcTask Outputs/GVL_iXlinker.EtherCAT_Master_ERxxxx.Beckhoff_ER2xxx.Beckhoff_ER2xxxEK1122.A_0036_ER2339_0021_0018.Channel_22.Output <-> Channel 22/Output
//     PlcTask Outputs/GVL_iXlinker.EtherCAT_Master_ERxxxx.Beckhoff_ER2xxx.Beckhoff_ER2xxxEK1122.A_0036_ER2339_0021_0018.Channel_23.Output <-> Channel 23/Output
//     PlcTask Outputs/GVL_iXlinker.EtherCAT_Master_ERxxxx.Beckhoff_ER2xxx.Beckhoff_ER2xxxEK1122.A_0036_ER2339_0021_0018.Channel_24.Output <-> Channel 24/Output
//     PlcTask Outputs/GVL_iXlinker.EtherCAT_Master_ERxxxx.Beckhoff_ER2xxx.Beckhoff_ER2xxxEK1122.A_0036_ER2339_0021_0018.Channel_25.Output <-> Channel 25/Output
//     PlcTask Outputs/GVL_iXlinker.EtherCAT_Master_ERxxxx.Beckhoff_ER2xxx.Beckhoff_ER2xxxEK1122.A_0036_ER2339_0021_0018.Channel_26.Output <-> Channel 26/Output
//     PlcTask Outputs/GVL_iXlinker.EtherCAT_Master_ERxxxx.Beckhoff_ER2xxx.Beckhoff_ER2xxxEK1122.A_0036_ER2339_0021_0018.Channel_27.Output <-> Channel 27/Output
//     PlcTask Outputs/GVL_iXlinker.EtherCAT_Master_ERxxxx.Beckhoff_ER2xxx.Beckhoff_ER2xxxEK1122.A_0036_ER2339_0021_0018.Channel_28.Output <-> Channel 28/Output
//     PlcTask Outputs/GVL_iXlinker.EtherCAT_Master_ERxxxx.Beckhoff_ER2xxx.Beckhoff_ER2xxxEK1122.A_0036_ER2339_0021_0018.Channel_29.Output <-> Channel 29/Output
//     PlcTask Outputs/GVL_iXlinker.EtherCAT_Master_ERxxxx.Beckhoff_ER2xxx.Beckhoff_ER2xxxEK1122.A_0036_ER2339_0021_0018.Channel_30.Output <-> Channel 30/Output
//     PlcTask Outputs/GVL_iXlinker.EtherCAT_Master_ERxxxx.Beckhoff_ER2xxx.Beckhoff_ER2xxxEK1122.A_0036_ER2339_0021_0018.Channel_31.Output <-> Channel 31/Output
//     PlcTask Outputs/GVL_iXlinker.EtherCAT_Master_ERxxxx.Beckhoff_ER2xxx.Beckhoff_ER2xxxEK1122.A_0036_ER2339_0021_0018.Channel_32.Output <-> Channel 32/Output
//     PlcTask Inputs/GVL_iXlinker.EtherCAT_Master_ERxxxx.Beckhoff_ER2xxx.Beckhoff_ER2xxxEK1122.A_0036_ER2339_0021_0018.WcState.WcState <-> WcState/WcState
//     PlcTask Inputs/GVL_iXlinker.EtherCAT_Master_ERxxxx.Beckhoff_ER2xxx.Beckhoff_ER2xxxEK1122.A_0036_ER2339_0021_0018.WcState.InputToggle <-> WcState/InputToggle
//     PlcTask Inputs/GVL_iXlinker.EtherCAT_Master_ERxxxx.Beckhoff_ER2xxx.Beckhoff_ER2xxxEK1122.A_0036_ER2339_0021_0018.InfoData.AoeNetId <-> InfoData/AoeNetId
//     PlcTask Inputs/GVL_iXlinker.EtherCAT_Master_ERxxxx.Beckhoff_ER2xxx.Beckhoff_ER2xxxEK1122.A_0036_ER2339_0021_0018.InfoData.State <-> InfoData/State
//   PLC/PLC Instance <-> EtherCAT Master ERxxxx/Beckhoff ER2xxx/Beckhoff ER2xxxEK1122/A_0037(ER2339-0021-0019)
//     PlcTask Inputs/GVL_iXlinker.EtherCAT_Master_ERxxxx.Beckhoff_ER2xxx.Beckhoff_ER2xxxEK1122.A_0037_ER2339_0021_0019.Channel_1.Input <-> Channel 1/Input
//     PlcTask Inputs/GVL_iXlinker.EtherCAT_Master_ERxxxx.Beckhoff_ER2xxx.Beckhoff_ER2xxxEK1122.A_0037_ER2339_0021_0019.Channel_2.Input <-> Channel 2/Input
//     PlcTask Inputs/GVL_iXlinker.EtherCAT_Master_ERxxxx.Beckhoff_ER2xxx.Beckhoff_ER2xxxEK1122.A_0037_ER2339_0021_0019.Channel_3.Input <-> Channel 3/Input
//     PlcTask Inputs/GVL_iXlinker.EtherCAT_Master_ERxxxx.Beckhoff_ER2xxx.Beckhoff_ER2xxxEK1122.A_0037_ER2339_0021_0019.Channel_4.Input <-> Channel 4/Input
//     PlcTask Inputs/GVL_iXlinker.EtherCAT_Master_ERxxxx.Beckhoff_ER2xxx.Beckhoff_ER2xxxEK1122.A_0037_ER2339_0021_0019.Channel_5.Input <-> Channel 5/Input
//     PlcTask Inputs/GVL_iXlinker.EtherCAT_Master_ERxxxx.Beckhoff_ER2xxx.Beckhoff_ER2xxxEK1122.A_0037_ER2339_0021_0019.Channel_6.Input <-> Channel 6/Input
//     PlcTask Inputs/GVL_iXlinker.EtherCAT_Master_ERxxxx.Beckhoff_ER2xxx.Beckhoff_ER2xxxEK1122.A_0037_ER2339_0021_0019.Channel_7.Input <-> Channel 7/Input
//     PlcTask Inputs/GVL_iXlinker.EtherCAT_Master_ERxxxx.Beckhoff_ER2xxx.Beckhoff_ER2xxxEK1122.A_0037_ER2339_0021_0019.Channel_8.Input <-> Channel 8/Input
//     PlcTask Inputs/GVL_iXlinker.EtherCAT_Master_ERxxxx.Beckhoff_ER2xxx.Beckhoff_ER2xxxEK1122.A_0037_ER2339_0021_0019.Channel_9.Input <-> Channel 9/Input
//     PlcTask Inputs/GVL_iXlinker.EtherCAT_Master_ERxxxx.Beckhoff_ER2xxx.Beckhoff_ER2xxxEK1122.A_0037_ER2339_0021_0019.Channel_10.Input <-> Channel 10/Input
//     PlcTask Inputs/GVL_iXlinker.EtherCAT_Master_ERxxxx.Beckhoff_ER2xxx.Beckhoff_ER2xxxEK1122.A_0037_ER2339_0021_0019.Channel_11.Input <-> Channel 11/Input
//     PlcTask Inputs/GVL_iXlinker.EtherCAT_Master_ERxxxx.Beckhoff_ER2xxx.Beckhoff_ER2xxxEK1122.A_0037_ER2339_0021_0019.Channel_12.Input <-> Channel 12/Input
//     PlcTask Inputs/GVL_iXlinker.EtherCAT_Master_ERxxxx.Beckhoff_ER2xxx.Beckhoff_ER2xxxEK1122.A_0037_ER2339_0021_0019.Channel_13.Input <-> Channel 13/Input
//     PlcTask Inputs/GVL_iXlinker.EtherCAT_Master_ERxxxx.Beckhoff_ER2xxx.Beckhoff_ER2xxxEK1122.A_0037_ER2339_0021_0019.Channel_14.Input <-> Channel 14/Input
//     PlcTask Inputs/GVL_iXlinker.EtherCAT_Master_ERxxxx.Beckhoff_ER2xxx.Beckhoff_ER2xxxEK1122.A_0037_ER2339_0021_0019.Channel_15.Input <-> Channel 15/Input
//     PlcTask Inputs/GVL_iXlinker.EtherCAT_Master_ERxxxx.Beckhoff_ER2xxx.Beckhoff_ER2xxxEK1122.A_0037_ER2339_0021_0019.Channel_16.Input <-> Channel 16/Input
//     PlcTask Outputs/GVL_iXlinker.EtherCAT_Master_ERxxxx.Beckhoff_ER2xxx.Beckhoff_ER2xxxEK1122.A_0037_ER2339_0021_0019.Channel_17.Output <-> Channel 17/Output
//     PlcTask Outputs/GVL_iXlinker.EtherCAT_Master_ERxxxx.Beckhoff_ER2xxx.Beckhoff_ER2xxxEK1122.A_0037_ER2339_0021_0019.Channel_18.Output <-> Channel 18/Output
//     PlcTask Outputs/GVL_iXlinker.EtherCAT_Master_ERxxxx.Beckhoff_ER2xxx.Beckhoff_ER2xxxEK1122.A_0037_ER2339_0021_0019.Channel_19.Output <-> Channel 19/Output
//     PlcTask Outputs/GVL_iXlinker.EtherCAT_Master_ERxxxx.Beckhoff_ER2xxx.Beckhoff_ER2xxxEK1122.A_0037_ER2339_0021_0019.Channel_20.Output <-> Channel 20/Output
//     PlcTask Outputs/GVL_iXlinker.EtherCAT_Master_ERxxxx.Beckhoff_ER2xxx.Beckhoff_ER2xxxEK1122.A_0037_ER2339_0021_0019.Channel_21.Output <-> Channel 21/Output
//     PlcTask Outputs/GVL_iXlinker.EtherCAT_Master_ERxxxx.Beckhoff_ER2xxx.Beckhoff_ER2xxxEK1122.A_0037_ER2339_0021_0019.Channel_22.Output <-> Channel 22/Output
//     PlcTask Outputs/GVL_iXlinker.EtherCAT_Master_ERxxxx.Beckhoff_ER2xxx.Beckhoff_ER2xxxEK1122.A_0037_ER2339_0021_0019.Channel_23.Output <-> Channel 23/Output
//     PlcTask Outputs/GVL_iXlinker.EtherCAT_Master_ERxxxx.Beckhoff_ER2xxx.Beckhoff_ER2xxxEK1122.A_0037_ER2339_0021_0019.Channel_24.Output <-> Channel 24/Output
//     PlcTask Outputs/GVL_iXlinker.EtherCAT_Master_ERxxxx.Beckhoff_ER2xxx.Beckhoff_ER2xxxEK1122.A_0037_ER2339_0021_0019.Channel_25.Output <-> Channel 25/Output
//     PlcTask Outputs/GVL_iXlinker.EtherCAT_Master_ERxxxx.Beckhoff_ER2xxx.Beckhoff_ER2xxxEK1122.A_0037_ER2339_0021_0019.Channel_26.Output <-> Channel 26/Output
//     PlcTask Outputs/GVL_iXlinker.EtherCAT_Master_ERxxxx.Beckhoff_ER2xxx.Beckhoff_ER2xxxEK1122.A_0037_ER2339_0021_0019.Channel_27.Output <-> Channel 27/Output
//     PlcTask Outputs/GVL_iXlinker.EtherCAT_Master_ERxxxx.Beckhoff_ER2xxx.Beckhoff_ER2xxxEK1122.A_0037_ER2339_0021_0019.Channel_28.Output <-> Channel 28/Output
//     PlcTask Outputs/GVL_iXlinker.EtherCAT_Master_ERxxxx.Beckhoff_ER2xxx.Beckhoff_ER2xxxEK1122.A_0037_ER2339_0021_0019.Channel_29.Output <-> Channel 29/Output
//     PlcTask Outputs/GVL_iXlinker.EtherCAT_Master_ERxxxx.Beckhoff_ER2xxx.Beckhoff_ER2xxxEK1122.A_0037_ER2339_0021_0019.Channel_30.Output <-> Channel 30/Output
//     PlcTask Outputs/GVL_iXlinker.EtherCAT_Master_ERxxxx.Beckhoff_ER2xxx.Beckhoff_ER2xxxEK1122.A_0037_ER2339_0021_0019.Channel_31.Output <-> Channel 31/Output
//     PlcTask Outputs/GVL_iXlinker.EtherCAT_Master_ERxxxx.Beckhoff_ER2xxx.Beckhoff_ER2xxxEK1122.A_0037_ER2339_0021_0019.Channel_32.Output <-> Channel 32/Output
//     PlcTask Inputs/GVL_iXlinker.EtherCAT_Master_ERxxxx.Beckhoff_ER2xxx.Beckhoff_ER2xxxEK1122.A_0037_ER2339_0021_0019.WcState.WcState <-> WcState/WcState
//     PlcTask Inputs/GVL_iXlinker.EtherCAT_Master_ERxxxx.Beckhoff_ER2xxx.Beckhoff_ER2xxxEK1122.A_0037_ER2339_0021_0019.WcState.InputToggle <-> WcState/InputToggle
//     PlcTask Inputs/GVL_iXlinker.EtherCAT_Master_ERxxxx.Beckhoff_ER2xxx.Beckhoff_ER2xxxEK1122.A_0037_ER2339_0021_0019.InfoData.State <-> InfoData/State
//   PLC/PLC Instance <-> EtherCAT Master ERxxxx/Beckhoff ER2xxx/Beckhoff ER2xxxEK1122/A_0038(ER2339-0022-0018)
//     PlcTask Inputs/GVL_iXlinker.EtherCAT_Master_ERxxxx.Beckhoff_ER2xxx.Beckhoff_ER2xxxEK1122.A_0038_ER2339_0022_0018.Channel_1.Input <-> Channel 1/Input
//     PlcTask Inputs/GVL_iXlinker.EtherCAT_Master_ERxxxx.Beckhoff_ER2xxx.Beckhoff_ER2xxxEK1122.A_0038_ER2339_0022_0018.Channel_2.Input <-> Channel 2/Input
//     PlcTask Inputs/GVL_iXlinker.EtherCAT_Master_ERxxxx.Beckhoff_ER2xxx.Beckhoff_ER2xxxEK1122.A_0038_ER2339_0022_0018.Channel_3.Input <-> Channel 3/Input
//     PlcTask Inputs/GVL_iXlinker.EtherCAT_Master_ERxxxx.Beckhoff_ER2xxx.Beckhoff_ER2xxxEK1122.A_0038_ER2339_0022_0018.Channel_4.Input <-> Channel 4/Input
//     PlcTask Inputs/GVL_iXlinker.EtherCAT_Master_ERxxxx.Beckhoff_ER2xxx.Beckhoff_ER2xxxEK1122.A_0038_ER2339_0022_0018.Channel_5.Input <-> Channel 5/Input
//     PlcTask Inputs/GVL_iXlinker.EtherCAT_Master_ERxxxx.Beckhoff_ER2xxx.Beckhoff_ER2xxxEK1122.A_0038_ER2339_0022_0018.Channel_6.Input <-> Channel 6/Input
//     PlcTask Inputs/GVL_iXlinker.EtherCAT_Master_ERxxxx.Beckhoff_ER2xxx.Beckhoff_ER2xxxEK1122.A_0038_ER2339_0022_0018.Channel_7.Input <-> Channel 7/Input
//     PlcTask Inputs/GVL_iXlinker.EtherCAT_Master_ERxxxx.Beckhoff_ER2xxx.Beckhoff_ER2xxxEK1122.A_0038_ER2339_0022_0018.Channel_8.Input <-> Channel 8/Input
//     PlcTask Inputs/GVL_iXlinker.EtherCAT_Master_ERxxxx.Beckhoff_ER2xxx.Beckhoff_ER2xxxEK1122.A_0038_ER2339_0022_0018.Channel_9.Input <-> Channel 9/Input
//     PlcTask Inputs/GVL_iXlinker.EtherCAT_Master_ERxxxx.Beckhoff_ER2xxx.Beckhoff_ER2xxxEK1122.A_0038_ER2339_0022_0018.Channel_10.Input <-> Channel 10/Input
//     PlcTask Inputs/GVL_iXlinker.EtherCAT_Master_ERxxxx.Beckhoff_ER2xxx.Beckhoff_ER2xxxEK1122.A_0038_ER2339_0022_0018.Channel_11.Input <-> Channel 11/Input
//     PlcTask Inputs/GVL_iXlinker.EtherCAT_Master_ERxxxx.Beckhoff_ER2xxx.Beckhoff_ER2xxxEK1122.A_0038_ER2339_0022_0018.Channel_12.Input <-> Channel 12/Input
//     PlcTask Inputs/GVL_iXlinker.EtherCAT_Master_ERxxxx.Beckhoff_ER2xxx.Beckhoff_ER2xxxEK1122.A_0038_ER2339_0022_0018.Channel_13.Input <-> Channel 13/Input
//     PlcTask Inputs/GVL_iXlinker.EtherCAT_Master_ERxxxx.Beckhoff_ER2xxx.Beckhoff_ER2xxxEK1122.A_0038_ER2339_0022_0018.Channel_14.Input <-> Channel 14/Input
//     PlcTask Inputs/GVL_iXlinker.EtherCAT_Master_ERxxxx.Beckhoff_ER2xxx.Beckhoff_ER2xxxEK1122.A_0038_ER2339_0022_0018.Channel_15.Input <-> Channel 15/Input
//     PlcTask Inputs/GVL_iXlinker.EtherCAT_Master_ERxxxx.Beckhoff_ER2xxx.Beckhoff_ER2xxxEK1122.A_0038_ER2339_0022_0018.Channel_16.Input <-> Channel 16/Input
//     PlcTask Outputs/GVL_iXlinker.EtherCAT_Master_ERxxxx.Beckhoff_ER2xxx.Beckhoff_ER2xxxEK1122.A_0038_ER2339_0022_0018.Channel_17.Output <-> Channel 17/Output
//     PlcTask Outputs/GVL_iXlinker.EtherCAT_Master_ERxxxx.Beckhoff_ER2xxx.Beckhoff_ER2xxxEK1122.A_0038_ER2339_0022_0018.Channel_18.Output <-> Channel 18/Output
//     PlcTask Outputs/GVL_iXlinker.EtherCAT_Master_ERxxxx.Beckhoff_ER2xxx.Beckhoff_ER2xxxEK1122.A_0038_ER2339_0022_0018.Channel_19.Output <-> Channel 19/Output
//     PlcTask Outputs/GVL_iXlinker.EtherCAT_Master_ERxxxx.Beckhoff_ER2xxx.Beckhoff_ER2xxxEK1122.A_0038_ER2339_0022_0018.Channel_20.Output <-> Channel 20/Output
//     PlcTask Outputs/GVL_iXlinker.EtherCAT_Master_ERxxxx.Beckhoff_ER2xxx.Beckhoff_ER2xxxEK1122.A_0038_ER2339_0022_0018.Channel_21.Output <-> Channel 21/Output
//     PlcTask Outputs/GVL_iXlinker.EtherCAT_Master_ERxxxx.Beckhoff_ER2xxx.Beckhoff_ER2xxxEK1122.A_0038_ER2339_0022_0018.Channel_22.Output <-> Channel 22/Output
//     PlcTask Outputs/GVL_iXlinker.EtherCAT_Master_ERxxxx.Beckhoff_ER2xxx.Beckhoff_ER2xxxEK1122.A_0038_ER2339_0022_0018.Channel_23.Output <-> Channel 23/Output
//     PlcTask Outputs/GVL_iXlinker.EtherCAT_Master_ERxxxx.Beckhoff_ER2xxx.Beckhoff_ER2xxxEK1122.A_0038_ER2339_0022_0018.Channel_24.Output <-> Channel 24/Output
//     PlcTask Outputs/GVL_iXlinker.EtherCAT_Master_ERxxxx.Beckhoff_ER2xxx.Beckhoff_ER2xxxEK1122.A_0038_ER2339_0022_0018.Channel_25.Output <-> Channel 25/Output
//     PlcTask Outputs/GVL_iXlinker.EtherCAT_Master_ERxxxx.Beckhoff_ER2xxx.Beckhoff_ER2xxxEK1122.A_0038_ER2339_0022_0018.Channel_26.Output <-> Channel 26/Output
//     PlcTask Outputs/GVL_iXlinker.EtherCAT_Master_ERxxxx.Beckhoff_ER2xxx.Beckhoff_ER2xxxEK1122.A_0038_ER2339_0022_0018.Channel_27.Output <-> Channel 27/Output
//     PlcTask Outputs/GVL_iXlinker.EtherCAT_Master_ERxxxx.Beckhoff_ER2xxx.Beckhoff_ER2xxxEK1122.A_0038_ER2339_0022_0018.Channel_28.Output <-> Channel 28/Output
//     PlcTask Outputs/GVL_iXlinker.EtherCAT_Master_ERxxxx.Beckhoff_ER2xxx.Beckhoff_ER2xxxEK1122.A_0038_ER2339_0022_0018.Channel_29.Output <-> Channel 29/Output
//     PlcTask Outputs/GVL_iXlinker.EtherCAT_Master_ERxxxx.Beckhoff_ER2xxx.Beckhoff_ER2xxxEK1122.A_0038_ER2339_0022_0018.Channel_30.Output <-> Channel 30/Output
//     PlcTask Outputs/GVL_iXlinker.EtherCAT_Master_ERxxxx.Beckhoff_ER2xxx.Beckhoff_ER2xxxEK1122.A_0038_ER2339_0022_0018.Channel_31.Output <-> Channel 31/Output
//     PlcTask Outputs/GVL_iXlinker.EtherCAT_Master_ERxxxx.Beckhoff_ER2xxx.Beckhoff_ER2xxxEK1122.A_0038_ER2339_0022_0018.Channel_32.Output <-> Channel 32/Output
//     PlcTask Inputs/GVL_iXlinker.EtherCAT_Master_ERxxxx.Beckhoff_ER2xxx.Beckhoff_ER2xxxEK1122.A_0038_ER2339_0022_0018.WcState.WcState <-> WcState/WcState
//     PlcTask Inputs/GVL_iXlinker.EtherCAT_Master_ERxxxx.Beckhoff_ER2xxx.Beckhoff_ER2xxxEK1122.A_0038_ER2339_0022_0018.WcState.InputToggle <-> WcState/InputToggle
//     PlcTask Inputs/GVL_iXlinker.EtherCAT_Master_ERxxxx.Beckhoff_ER2xxx.Beckhoff_ER2xxxEK1122.A_0038_ER2339_0022_0018.InfoData.State <-> InfoData/State
//   PLC/PLC Instance <-> EtherCAT Master ERxxxx/Beckhoff ER2xxx/Beckhoff ER2xxxEK1122/A_0039(ER2339-0022-0019)
//     PlcTask Inputs/GVL_iXlinker.EtherCAT_Master_ERxxxx.Beckhoff_ER2xxx.Beckhoff_ER2xxxEK1122.A_0039_ER2339_0022_0019.Channel_1.Input <-> Channel 1/Input
//     PlcTask Inputs/GVL_iXlinker.EtherCAT_Master_ERxxxx.Beckhoff_ER2xxx.Beckhoff_ER2xxxEK1122.A_0039_ER2339_0022_0019.Channel_2.Input <-> Channel 2/Input
//     PlcTask Inputs/GVL_iXlinker.EtherCAT_Master_ERxxxx.Beckhoff_ER2xxx.Beckhoff_ER2xxxEK1122.A_0039_ER2339_0022_0019.Channel_3.Input <-> Channel 3/Input
//     PlcTask Inputs/GVL_iXlinker.EtherCAT_Master_ERxxxx.Beckhoff_ER2xxx.Beckhoff_ER2xxxEK1122.A_0039_ER2339_0022_0019.Channel_4.Input <-> Channel 4/Input
//     PlcTask Inputs/GVL_iXlinker.EtherCAT_Master_ERxxxx.Beckhoff_ER2xxx.Beckhoff_ER2xxxEK1122.A_0039_ER2339_0022_0019.Channel_5.Input <-> Channel 5/Input
//     PlcTask Inputs/GVL_iXlinker.EtherCAT_Master_ERxxxx.Beckhoff_ER2xxx.Beckhoff_ER2xxxEK1122.A_0039_ER2339_0022_0019.Channel_6.Input <-> Channel 6/Input
//     PlcTask Inputs/GVL_iXlinker.EtherCAT_Master_ERxxxx.Beckhoff_ER2xxx.Beckhoff_ER2xxxEK1122.A_0039_ER2339_0022_0019.Channel_7.Input <-> Channel 7/Input
//     PlcTask Inputs/GVL_iXlinker.EtherCAT_Master_ERxxxx.Beckhoff_ER2xxx.Beckhoff_ER2xxxEK1122.A_0039_ER2339_0022_0019.Channel_8.Input <-> Channel 8/Input
//     PlcTask Inputs/GVL_iXlinker.EtherCAT_Master_ERxxxx.Beckhoff_ER2xxx.Beckhoff_ER2xxxEK1122.A_0039_ER2339_0022_0019.Channel_9.Input <-> Channel 9/Input
//     PlcTask Inputs/GVL_iXlinker.EtherCAT_Master_ERxxxx.Beckhoff_ER2xxx.Beckhoff_ER2xxxEK1122.A_0039_ER2339_0022_0019.Channel_10.Input <-> Channel 10/Input
//     PlcTask Inputs/GVL_iXlinker.EtherCAT_Master_ERxxxx.Beckhoff_ER2xxx.Beckhoff_ER2xxxEK1122.A_0039_ER2339_0022_0019.Channel_11.Input <-> Channel 11/Input
//     PlcTask Inputs/GVL_iXlinker.EtherCAT_Master_ERxxxx.Beckhoff_ER2xxx.Beckhoff_ER2xxxEK1122.A_0039_ER2339_0022_0019.Channel_12.Input <-> Channel 12/Input
//     PlcTask Inputs/GVL_iXlinker.EtherCAT_Master_ERxxxx.Beckhoff_ER2xxx.Beckhoff_ER2xxxEK1122.A_0039_ER2339_0022_0019.Channel_13.Input <-> Channel 13/Input
//     PlcTask Inputs/GVL_iXlinker.EtherCAT_Master_ERxxxx.Beckhoff_ER2xxx.Beckhoff_ER2xxxEK1122.A_0039_ER2339_0022_0019.Channel_14.Input <-> Channel 14/Input
//     PlcTask Inputs/GVL_iXlinker.EtherCAT_Master_ERxxxx.Beckhoff_ER2xxx.Beckhoff_ER2xxxEK1122.A_0039_ER2339_0022_0019.Channel_15.Input <-> Channel 15/Input
//     PlcTask Inputs/GVL_iXlinker.EtherCAT_Master_ERxxxx.Beckhoff_ER2xxx.Beckhoff_ER2xxxEK1122.A_0039_ER2339_0022_0019.Channel_16.Input <-> Channel 16/Input
//     PlcTask Outputs/GVL_iXlinker.EtherCAT_Master_ERxxxx.Beckhoff_ER2xxx.Beckhoff_ER2xxxEK1122.A_0039_ER2339_0022_0019.Channel_17.Output <-> Channel 17/Output
//     PlcTask Outputs/GVL_iXlinker.EtherCAT_Master_ERxxxx.Beckhoff_ER2xxx.Beckhoff_ER2xxxEK1122.A_0039_ER2339_0022_0019.Channel_18.Output <-> Channel 18/Output
//     PlcTask Outputs/GVL_iXlinker.EtherCAT_Master_ERxxxx.Beckhoff_ER2xxx.Beckhoff_ER2xxxEK1122.A_0039_ER2339_0022_0019.Channel_19.Output <-> Channel 19/Output
//     PlcTask Outputs/GVL_iXlinker.EtherCAT_Master_ERxxxx.Beckhoff_ER2xxx.Beckhoff_ER2xxxEK1122.A_0039_ER2339_0022_0019.Channel_20.Output <-> Channel 20/Output
//     PlcTask Outputs/GVL_iXlinker.EtherCAT_Master_ERxxxx.Beckhoff_ER2xxx.Beckhoff_ER2xxxEK1122.A_0039_ER2339_0022_0019.Channel_21.Output <-> Channel 21/Output
//     PlcTask Outputs/GVL_iXlinker.EtherCAT_Master_ERxxxx.Beckhoff_ER2xxx.Beckhoff_ER2xxxEK1122.A_0039_ER2339_0022_0019.Channel_22.Output <-> Channel 22/Output
//     PlcTask Outputs/GVL_iXlinker.EtherCAT_Master_ERxxxx.Beckhoff_ER2xxx.Beckhoff_ER2xxxEK1122.A_0039_ER2339_0022_0019.Channel_23.Output <-> Channel 23/Output
//     PlcTask Outputs/GVL_iXlinker.EtherCAT_Master_ERxxxx.Beckhoff_ER2xxx.Beckhoff_ER2xxxEK1122.A_0039_ER2339_0022_0019.Channel_24.Output <-> Channel 24/Output
//     PlcTask Outputs/GVL_iXlinker.EtherCAT_Master_ERxxxx.Beckhoff_ER2xxx.Beckhoff_ER2xxxEK1122.A_0039_ER2339_0022_0019.Channel_25.Output <-> Channel 25/Output
//     PlcTask Outputs/GVL_iXlinker.EtherCAT_Master_ERxxxx.Beckhoff_ER2xxx.Beckhoff_ER2xxxEK1122.A_0039_ER2339_0022_0019.Channel_26.Output <-> Channel 26/Output
//     PlcTask Outputs/GVL_iXlinker.EtherCAT_Master_ERxxxx.Beckhoff_ER2xxx.Beckhoff_ER2xxxEK1122.A_0039_ER2339_0022_0019.Channel_27.Output <-> Channel 27/Output
//     PlcTask Outputs/GVL_iXlinker.EtherCAT_Master_ERxxxx.Beckhoff_ER2xxx.Beckhoff_ER2xxxEK1122.A_0039_ER2339_0022_0019.Channel_28.Output <-> Channel 28/Output
//     PlcTask Outputs/GVL_iXlinker.EtherCAT_Master_ERxxxx.Beckhoff_ER2xxx.Beckhoff_ER2xxxEK1122.A_0039_ER2339_0022_0019.Channel_29.Output <-> Channel 29/Output
//     PlcTask Outputs/GVL_iXlinker.EtherCAT_Master_ERxxxx.Beckhoff_ER2xxx.Beckhoff_ER2xxxEK1122.A_0039_ER2339_0022_0019.Channel_30.Output <-> Channel 30/Output
//     PlcTask Outputs/GVL_iXlinker.EtherCAT_Master_ERxxxx.Beckhoff_ER2xxx.Beckhoff_ER2xxxEK1122.A_0039_ER2339_0022_0019.Channel_31.Output <-> Channel 31/Output
//     PlcTask Outputs/GVL_iXlinker.EtherCAT_Master_ERxxxx.Beckhoff_ER2xxx.Beckhoff_ER2xxxEK1122.A_0039_ER2339_0022_0019.Channel_32.Output <-> Channel 32/Output
//     PlcTask Inputs/GVL_iXlinker.EtherCAT_Master_ERxxxx.Beckhoff_ER2xxx.Beckhoff_ER2xxxEK1122.A_0039_ER2339_0022_0019.WcState.WcState <-> WcState/WcState
//     PlcTask Inputs/GVL_iXlinker.EtherCAT_Master_ERxxxx.Beckhoff_ER2xxx.Beckhoff_ER2xxxEK1122.A_0039_ER2339_0022_0019.WcState.InputToggle <-> WcState/InputToggle
//     PlcTask Inputs/GVL_iXlinker.EtherCAT_Master_ERxxxx.Beckhoff_ER2xxx.Beckhoff_ER2xxxEK1122.A_0039_ER2339_0022_0019.InfoData.State <-> InfoData/State
//   PLC/PLC Instance <-> EtherCAT Master ERxxxx/Beckhoff ER2xxx/Beckhoff ER2xxxEK1122/A_0040(ER2349-0021-0017)
//     PlcTask Inputs/GVL_iXlinker.EtherCAT_Master_ERxxxx.Beckhoff_ER2xxx.Beckhoff_ER2xxxEK1122.A_0040_ER2349_0021_0017.Channel_1.Input <-> Channel 1/Input
//     PlcTask Inputs/GVL_iXlinker.EtherCAT_Master_ERxxxx.Beckhoff_ER2xxx.Beckhoff_ER2xxxEK1122.A_0040_ER2349_0021_0017.Channel_2.Input <-> Channel 2/Input
//     PlcTask Inputs/GVL_iXlinker.EtherCAT_Master_ERxxxx.Beckhoff_ER2xxx.Beckhoff_ER2xxxEK1122.A_0040_ER2349_0021_0017.Channel_3.Input <-> Channel 3/Input
//     PlcTask Inputs/GVL_iXlinker.EtherCAT_Master_ERxxxx.Beckhoff_ER2xxx.Beckhoff_ER2xxxEK1122.A_0040_ER2349_0021_0017.Channel_4.Input <-> Channel 4/Input
//     PlcTask Inputs/GVL_iXlinker.EtherCAT_Master_ERxxxx.Beckhoff_ER2xxx.Beckhoff_ER2xxxEK1122.A_0040_ER2349_0021_0017.Channel_5.Input <-> Channel 5/Input
//     PlcTask Inputs/GVL_iXlinker.EtherCAT_Master_ERxxxx.Beckhoff_ER2xxx.Beckhoff_ER2xxxEK1122.A_0040_ER2349_0021_0017.Channel_6.Input <-> Channel 6/Input
//     PlcTask Inputs/GVL_iXlinker.EtherCAT_Master_ERxxxx.Beckhoff_ER2xxx.Beckhoff_ER2xxxEK1122.A_0040_ER2349_0021_0017.Channel_7.Input <-> Channel 7/Input
//     PlcTask Inputs/GVL_iXlinker.EtherCAT_Master_ERxxxx.Beckhoff_ER2xxx.Beckhoff_ER2xxxEK1122.A_0040_ER2349_0021_0017.Channel_8.Input <-> Channel 8/Input
//     PlcTask Inputs/GVL_iXlinker.EtherCAT_Master_ERxxxx.Beckhoff_ER2xxx.Beckhoff_ER2xxxEK1122.A_0040_ER2349_0021_0017.Channel_9.Input <-> Channel 9/Input
//     PlcTask Inputs/GVL_iXlinker.EtherCAT_Master_ERxxxx.Beckhoff_ER2xxx.Beckhoff_ER2xxxEK1122.A_0040_ER2349_0021_0017.Channel_10.Input <-> Channel 10/Input
//     PlcTask Inputs/GVL_iXlinker.EtherCAT_Master_ERxxxx.Beckhoff_ER2xxx.Beckhoff_ER2xxxEK1122.A_0040_ER2349_0021_0017.Channel_11.Input <-> Channel 11/Input
//     PlcTask Inputs/GVL_iXlinker.EtherCAT_Master_ERxxxx.Beckhoff_ER2xxx.Beckhoff_ER2xxxEK1122.A_0040_ER2349_0021_0017.Channel_12.Input <-> Channel 12/Input
//     PlcTask Inputs/GVL_iXlinker.EtherCAT_Master_ERxxxx.Beckhoff_ER2xxx.Beckhoff_ER2xxxEK1122.A_0040_ER2349_0021_0017.Channel_13.Input <-> Channel 13/Input
//     PlcTask Inputs/GVL_iXlinker.EtherCAT_Master_ERxxxx.Beckhoff_ER2xxx.Beckhoff_ER2xxxEK1122.A_0040_ER2349_0021_0017.Channel_14.Input <-> Channel 14/Input
//     PlcTask Inputs/GVL_iXlinker.EtherCAT_Master_ERxxxx.Beckhoff_ER2xxx.Beckhoff_ER2xxxEK1122.A_0040_ER2349_0021_0017.Channel_15.Input <-> Channel 15/Input
//     PlcTask Inputs/GVL_iXlinker.EtherCAT_Master_ERxxxx.Beckhoff_ER2xxx.Beckhoff_ER2xxxEK1122.A_0040_ER2349_0021_0017.Channel_16.Input <-> Channel 16/Input
//     PlcTask Outputs/GVL_iXlinker.EtherCAT_Master_ERxxxx.Beckhoff_ER2xxx.Beckhoff_ER2xxxEK1122.A_0040_ER2349_0021_0017.Channel_17.Output <-> Channel 17/Output
//     PlcTask Outputs/GVL_iXlinker.EtherCAT_Master_ERxxxx.Beckhoff_ER2xxx.Beckhoff_ER2xxxEK1122.A_0040_ER2349_0021_0017.Channel_18.Output <-> Channel 18/Output
//     PlcTask Outputs/GVL_iXlinker.EtherCAT_Master_ERxxxx.Beckhoff_ER2xxx.Beckhoff_ER2xxxEK1122.A_0040_ER2349_0021_0017.Channel_19.Output <-> Channel 19/Output
//     PlcTask Outputs/GVL_iXlinker.EtherCAT_Master_ERxxxx.Beckhoff_ER2xxx.Beckhoff_ER2xxxEK1122.A_0040_ER2349_0021_0017.Channel_20.Output <-> Channel 20/Output
//     PlcTask Outputs/GVL_iXlinker.EtherCAT_Master_ERxxxx.Beckhoff_ER2xxx.Beckhoff_ER2xxxEK1122.A_0040_ER2349_0021_0017.Channel_21.Output <-> Channel 21/Output
//     PlcTask Outputs/GVL_iXlinker.EtherCAT_Master_ERxxxx.Beckhoff_ER2xxx.Beckhoff_ER2xxxEK1122.A_0040_ER2349_0021_0017.Channel_22.Output <-> Channel 22/Output
//     PlcTask Outputs/GVL_iXlinker.EtherCAT_Master_ERxxxx.Beckhoff_ER2xxx.Beckhoff_ER2xxxEK1122.A_0040_ER2349_0021_0017.Channel_23.Output <-> Channel 23/Output
//     PlcTask Outputs/GVL_iXlinker.EtherCAT_Master_ERxxxx.Beckhoff_ER2xxx.Beckhoff_ER2xxxEK1122.A_0040_ER2349_0021_0017.Channel_24.Output <-> Channel 24/Output
//     PlcTask Outputs/GVL_iXlinker.EtherCAT_Master_ERxxxx.Beckhoff_ER2xxx.Beckhoff_ER2xxxEK1122.A_0040_ER2349_0021_0017.Channel_25.Output <-> Channel 25/Output
//     PlcTask Outputs/GVL_iXlinker.EtherCAT_Master_ERxxxx.Beckhoff_ER2xxx.Beckhoff_ER2xxxEK1122.A_0040_ER2349_0021_0017.Channel_26.Output <-> Channel 26/Output
//     PlcTask Outputs/GVL_iXlinker.EtherCAT_Master_ERxxxx.Beckhoff_ER2xxx.Beckhoff_ER2xxxEK1122.A_0040_ER2349_0021_0017.Channel_27.Output <-> Channel 27/Output
//     PlcTask Outputs/GVL_iXlinker.EtherCAT_Master_ERxxxx.Beckhoff_ER2xxx.Beckhoff_ER2xxxEK1122.A_0040_ER2349_0021_0017.Channel_28.Output <-> Channel 28/Output
//     PlcTask Outputs/GVL_iXlinker.EtherCAT_Master_ERxxxx.Beckhoff_ER2xxx.Beckhoff_ER2xxxEK1122.A_0040_ER2349_0021_0017.Channel_29.Output <-> Channel 29/Output
//     PlcTask Outputs/GVL_iXlinker.EtherCAT_Master_ERxxxx.Beckhoff_ER2xxx.Beckhoff_ER2xxxEK1122.A_0040_ER2349_0021_0017.Channel_30.Output <-> Channel 30/Output
//     PlcTask Outputs/GVL_iXlinker.EtherCAT_Master_ERxxxx.Beckhoff_ER2xxx.Beckhoff_ER2xxxEK1122.A_0040_ER2349_0021_0017.Channel_31.Output <-> Channel 31/Output
//     PlcTask Outputs/GVL_iXlinker.EtherCAT_Master_ERxxxx.Beckhoff_ER2xxx.Beckhoff_ER2xxxEK1122.A_0040_ER2349_0021_0017.Channel_32.Output <-> Channel 32/Output
//     PlcTask Inputs/GVL_iXlinker.EtherCAT_Master_ERxxxx.Beckhoff_ER2xxx.Beckhoff_ER2xxxEK1122.A_0040_ER2349_0021_0017.WcState.WcState <-> WcState/WcState
//     PlcTask Inputs/GVL_iXlinker.EtherCAT_Master_ERxxxx.Beckhoff_ER2xxx.Beckhoff_ER2xxxEK1122.A_0040_ER2349_0021_0017.WcState.InputToggle <-> WcState/InputToggle
//     PlcTask Inputs/GVL_iXlinker.EtherCAT_Master_ERxxxx.Beckhoff_ER2xxx.Beckhoff_ER2xxxEK1122.A_0040_ER2349_0021_0017.InfoData.State <-> InfoData/State
//   PLC/PLC Instance <-> EtherCAT Master ERxxxx/Beckhoff ER2xxx/Beckhoff ER2xxxEK1122/A_0041(ER2349-0021-0018)
//     PlcTask Inputs/GVL_iXlinker.EtherCAT_Master_ERxxxx.Beckhoff_ER2xxx.Beckhoff_ER2xxxEK1122.A_0041_ER2349_0021_0018.Channel_1.Input <-> Channel 1/Input
//     PlcTask Inputs/GVL_iXlinker.EtherCAT_Master_ERxxxx.Beckhoff_ER2xxx.Beckhoff_ER2xxxEK1122.A_0041_ER2349_0021_0018.Channel_2.Input <-> Channel 2/Input
//     PlcTask Inputs/GVL_iXlinker.EtherCAT_Master_ERxxxx.Beckhoff_ER2xxx.Beckhoff_ER2xxxEK1122.A_0041_ER2349_0021_0018.Channel_3.Input <-> Channel 3/Input
//     PlcTask Inputs/GVL_iXlinker.EtherCAT_Master_ERxxxx.Beckhoff_ER2xxx.Beckhoff_ER2xxxEK1122.A_0041_ER2349_0021_0018.Channel_4.Input <-> Channel 4/Input
//     PlcTask Inputs/GVL_iXlinker.EtherCAT_Master_ERxxxx.Beckhoff_ER2xxx.Beckhoff_ER2xxxEK1122.A_0041_ER2349_0021_0018.Channel_5.Input <-> Channel 5/Input
//     PlcTask Inputs/GVL_iXlinker.EtherCAT_Master_ERxxxx.Beckhoff_ER2xxx.Beckhoff_ER2xxxEK1122.A_0041_ER2349_0021_0018.Channel_6.Input <-> Channel 6/Input
//     PlcTask Inputs/GVL_iXlinker.EtherCAT_Master_ERxxxx.Beckhoff_ER2xxx.Beckhoff_ER2xxxEK1122.A_0041_ER2349_0021_0018.Channel_7.Input <-> Channel 7/Input
//     PlcTask Inputs/GVL_iXlinker.EtherCAT_Master_ERxxxx.Beckhoff_ER2xxx.Beckhoff_ER2xxxEK1122.A_0041_ER2349_0021_0018.Channel_8.Input <-> Channel 8/Input
//     PlcTask Inputs/GVL_iXlinker.EtherCAT_Master_ERxxxx.Beckhoff_ER2xxx.Beckhoff_ER2xxxEK1122.A_0041_ER2349_0021_0018.Channel_9.Input <-> Channel 9/Input
//     PlcTask Inputs/GVL_iXlinker.EtherCAT_Master_ERxxxx.Beckhoff_ER2xxx.Beckhoff_ER2xxxEK1122.A_0041_ER2349_0021_0018.Channel_10.Input <-> Channel 10/Input
//     PlcTask Inputs/GVL_iXlinker.EtherCAT_Master_ERxxxx.Beckhoff_ER2xxx.Beckhoff_ER2xxxEK1122.A_0041_ER2349_0021_0018.Channel_11.Input <-> Channel 11/Input
//     PlcTask Inputs/GVL_iXlinker.EtherCAT_Master_ERxxxx.Beckhoff_ER2xxx.Beckhoff_ER2xxxEK1122.A_0041_ER2349_0021_0018.Channel_12.Input <-> Channel 12/Input
//     PlcTask Inputs/GVL_iXlinker.EtherCAT_Master_ERxxxx.Beckhoff_ER2xxx.Beckhoff_ER2xxxEK1122.A_0041_ER2349_0021_0018.Channel_13.Input <-> Channel 13/Input
//     PlcTask Inputs/GVL_iXlinker.EtherCAT_Master_ERxxxx.Beckhoff_ER2xxx.Beckhoff_ER2xxxEK1122.A_0041_ER2349_0021_0018.Channel_14.Input <-> Channel 14/Input
//     PlcTask Inputs/GVL_iXlinker.EtherCAT_Master_ERxxxx.Beckhoff_ER2xxx.Beckhoff_ER2xxxEK1122.A_0041_ER2349_0021_0018.Channel_15.Input <-> Channel 15/Input
//     PlcTask Inputs/GVL_iXlinker.EtherCAT_Master_ERxxxx.Beckhoff_ER2xxx.Beckhoff_ER2xxxEK1122.A_0041_ER2349_0021_0018.Channel_16.Input <-> Channel 16/Input
//     PlcTask Outputs/GVL_iXlinker.EtherCAT_Master_ERxxxx.Beckhoff_ER2xxx.Beckhoff_ER2xxxEK1122.A_0041_ER2349_0021_0018.Channel_17.Output <-> Channel 17/Output
//     PlcTask Outputs/GVL_iXlinker.EtherCAT_Master_ERxxxx.Beckhoff_ER2xxx.Beckhoff_ER2xxxEK1122.A_0041_ER2349_0021_0018.Channel_18.Output <-> Channel 18/Output
//     PlcTask Outputs/GVL_iXlinker.EtherCAT_Master_ERxxxx.Beckhoff_ER2xxx.Beckhoff_ER2xxxEK1122.A_0041_ER2349_0021_0018.Channel_19.Output <-> Channel 19/Output
//     PlcTask Outputs/GVL_iXlinker.EtherCAT_Master_ERxxxx.Beckhoff_ER2xxx.Beckhoff_ER2xxxEK1122.A_0041_ER2349_0021_0018.Channel_20.Output <-> Channel 20/Output
//     PlcTask Outputs/GVL_iXlinker.EtherCAT_Master_ERxxxx.Beckhoff_ER2xxx.Beckhoff_ER2xxxEK1122.A_0041_ER2349_0021_0018.Channel_21.Output <-> Channel 21/Output
//     PlcTask Outputs/GVL_iXlinker.EtherCAT_Master_ERxxxx.Beckhoff_ER2xxx.Beckhoff_ER2xxxEK1122.A_0041_ER2349_0021_0018.Channel_22.Output <-> Channel 22/Output
//     PlcTask Outputs/GVL_iXlinker.EtherCAT_Master_ERxxxx.Beckhoff_ER2xxx.Beckhoff_ER2xxxEK1122.A_0041_ER2349_0021_0018.Channel_23.Output <-> Channel 23/Output
//     PlcTask Outputs/GVL_iXlinker.EtherCAT_Master_ERxxxx.Beckhoff_ER2xxx.Beckhoff_ER2xxxEK1122.A_0041_ER2349_0021_0018.Channel_24.Output <-> Channel 24/Output
//     PlcTask Outputs/GVL_iXlinker.EtherCAT_Master_ERxxxx.Beckhoff_ER2xxx.Beckhoff_ER2xxxEK1122.A_0041_ER2349_0021_0018.Channel_25.Output <-> Channel 25/Output
//     PlcTask Outputs/GVL_iXlinker.EtherCAT_Master_ERxxxx.Beckhoff_ER2xxx.Beckhoff_ER2xxxEK1122.A_0041_ER2349_0021_0018.Channel_26.Output <-> Channel 26/Output
//     PlcTask Outputs/GVL_iXlinker.EtherCAT_Master_ERxxxx.Beckhoff_ER2xxx.Beckhoff_ER2xxxEK1122.A_0041_ER2349_0021_0018.Channel_27.Output <-> Channel 27/Output
//     PlcTask Outputs/GVL_iXlinker.EtherCAT_Master_ERxxxx.Beckhoff_ER2xxx.Beckhoff_ER2xxxEK1122.A_0041_ER2349_0021_0018.Channel_28.Output <-> Channel 28/Output
//     PlcTask Outputs/GVL_iXlinker.EtherCAT_Master_ERxxxx.Beckhoff_ER2xxx.Beckhoff_ER2xxxEK1122.A_0041_ER2349_0021_0018.Channel_29.Output <-> Channel 29/Output
//     PlcTask Outputs/GVL_iXlinker.EtherCAT_Master_ERxxxx.Beckhoff_ER2xxx.Beckhoff_ER2xxxEK1122.A_0041_ER2349_0021_0018.Channel_30.Output <-> Channel 30/Output
//     PlcTask Outputs/GVL_iXlinker.EtherCAT_Master_ERxxxx.Beckhoff_ER2xxx.Beckhoff_ER2xxxEK1122.A_0041_ER2349_0021_0018.Channel_31.Output <-> Channel 31/Output
//     PlcTask Outputs/GVL_iXlinker.EtherCAT_Master_ERxxxx.Beckhoff_ER2xxx.Beckhoff_ER2xxxEK1122.A_0041_ER2349_0021_0018.Channel_32.Output <-> Channel 32/Output
//     PlcTask Inputs/GVL_iXlinker.EtherCAT_Master_ERxxxx.Beckhoff_ER2xxx.Beckhoff_ER2xxxEK1122.A_0041_ER2349_0021_0018.WcState.WcState <-> WcState/WcState
//     PlcTask Inputs/GVL_iXlinker.EtherCAT_Master_ERxxxx.Beckhoff_ER2xxx.Beckhoff_ER2xxxEK1122.A_0041_ER2349_0021_0018.WcState.InputToggle <-> WcState/InputToggle
//     PlcTask Inputs/GVL_iXlinker.EtherCAT_Master_ERxxxx.Beckhoff_ER2xxx.Beckhoff_ER2xxxEK1122.A_0041_ER2349_0021_0018.InfoData.State <-> InfoData/State
//   PLC/PLC Instance <-> EtherCAT Master ERxxxx/Beckhoff ER2xxx/Beckhoff ER2xxxEK1122/A_0042(ER2349-0022-0017)
//     PlcTask Inputs/GVL_iXlinker.EtherCAT_Master_ERxxxx.Beckhoff_ER2xxx.Beckhoff_ER2xxxEK1122.A_0042_ER2349_0022_0017.Channel_1.Input <-> Channel 1/Input
//     PlcTask Inputs/GVL_iXlinker.EtherCAT_Master_ERxxxx.Beckhoff_ER2xxx.Beckhoff_ER2xxxEK1122.A_0042_ER2349_0022_0017.Channel_2.Input <-> Channel 2/Input
//     PlcTask Inputs/GVL_iXlinker.EtherCAT_Master_ERxxxx.Beckhoff_ER2xxx.Beckhoff_ER2xxxEK1122.A_0042_ER2349_0022_0017.Channel_3.Input <-> Channel 3/Input
//     PlcTask Inputs/GVL_iXlinker.EtherCAT_Master_ERxxxx.Beckhoff_ER2xxx.Beckhoff_ER2xxxEK1122.A_0042_ER2349_0022_0017.Channel_4.Input <-> Channel 4/Input
//     PlcTask Inputs/GVL_iXlinker.EtherCAT_Master_ERxxxx.Beckhoff_ER2xxx.Beckhoff_ER2xxxEK1122.A_0042_ER2349_0022_0017.Channel_5.Input <-> Channel 5/Input
//     PlcTask Inputs/GVL_iXlinker.EtherCAT_Master_ERxxxx.Beckhoff_ER2xxx.Beckhoff_ER2xxxEK1122.A_0042_ER2349_0022_0017.Channel_6.Input <-> Channel 6/Input
//     PlcTask Inputs/GVL_iXlinker.EtherCAT_Master_ERxxxx.Beckhoff_ER2xxx.Beckhoff_ER2xxxEK1122.A_0042_ER2349_0022_0017.Channel_7.Input <-> Channel 7/Input
//     PlcTask Inputs/GVL_iXlinker.EtherCAT_Master_ERxxxx.Beckhoff_ER2xxx.Beckhoff_ER2xxxEK1122.A_0042_ER2349_0022_0017.Channel_8.Input <-> Channel 8/Input
//     PlcTask Inputs/GVL_iXlinker.EtherCAT_Master_ERxxxx.Beckhoff_ER2xxx.Beckhoff_ER2xxxEK1122.A_0042_ER2349_0022_0017.Channel_9.Input <-> Channel 9/Input
//     PlcTask Inputs/GVL_iXlinker.EtherCAT_Master_ERxxxx.Beckhoff_ER2xxx.Beckhoff_ER2xxxEK1122.A_0042_ER2349_0022_0017.Channel_10.Input <-> Channel 10/Input
//     PlcTask Inputs/GVL_iXlinker.EtherCAT_Master_ERxxxx.Beckhoff_ER2xxx.Beckhoff_ER2xxxEK1122.A_0042_ER2349_0022_0017.Channel_11.Input <-> Channel 11/Input
//     PlcTask Inputs/GVL_iXlinker.EtherCAT_Master_ERxxxx.Beckhoff_ER2xxx.Beckhoff_ER2xxxEK1122.A_0042_ER2349_0022_0017.Channel_12.Input <-> Channel 12/Input
//     PlcTask Inputs/GVL_iXlinker.EtherCAT_Master_ERxxxx.Beckhoff_ER2xxx.Beckhoff_ER2xxxEK1122.A_0042_ER2349_0022_0017.Channel_13.Input <-> Channel 13/Input
//     PlcTask Inputs/GVL_iXlinker.EtherCAT_Master_ERxxxx.Beckhoff_ER2xxx.Beckhoff_ER2xxxEK1122.A_0042_ER2349_0022_0017.Channel_14.Input <-> Channel 14/Input
//     PlcTask Inputs/GVL_iXlinker.EtherCAT_Master_ERxxxx.Beckhoff_ER2xxx.Beckhoff_ER2xxxEK1122.A_0042_ER2349_0022_0017.Channel_15.Input <-> Channel 15/Input
//     PlcTask Inputs/GVL_iXlinker.EtherCAT_Master_ERxxxx.Beckhoff_ER2xxx.Beckhoff_ER2xxxEK1122.A_0042_ER2349_0022_0017.Channel_16.Input <-> Channel 16/Input
//     PlcTask Outputs/GVL_iXlinker.EtherCAT_Master_ERxxxx.Beckhoff_ER2xxx.Beckhoff_ER2xxxEK1122.A_0042_ER2349_0022_0017.Channel_17.Output <-> Channel 17/Output
//     PlcTask Outputs/GVL_iXlinker.EtherCAT_Master_ERxxxx.Beckhoff_ER2xxx.Beckhoff_ER2xxxEK1122.A_0042_ER2349_0022_0017.Channel_18.Output <-> Channel 18/Output
//     PlcTask Outputs/GVL_iXlinker.EtherCAT_Master_ERxxxx.Beckhoff_ER2xxx.Beckhoff_ER2xxxEK1122.A_0042_ER2349_0022_0017.Channel_19.Output <-> Channel 19/Output
//     PlcTask Outputs/GVL_iXlinker.EtherCAT_Master_ERxxxx.Beckhoff_ER2xxx.Beckhoff_ER2xxxEK1122.A_0042_ER2349_0022_0017.Channel_20.Output <-> Channel 20/Output
//     PlcTask Outputs/GVL_iXlinker.EtherCAT_Master_ERxxxx.Beckhoff_ER2xxx.Beckhoff_ER2xxxEK1122.A_0042_ER2349_0022_0017.Channel_21.Output <-> Channel 21/Output
//     PlcTask Outputs/GVL_iXlinker.EtherCAT_Master_ERxxxx.Beckhoff_ER2xxx.Beckhoff_ER2xxxEK1122.A_0042_ER2349_0022_0017.Channel_22.Output <-> Channel 22/Output
//     PlcTask Outputs/GVL_iXlinker.EtherCAT_Master_ERxxxx.Beckhoff_ER2xxx.Beckhoff_ER2xxxEK1122.A_0042_ER2349_0022_0017.Channel_23.Output <-> Channel 23/Output
//     PlcTask Outputs/GVL_iXlinker.EtherCAT_Master_ERxxxx.Beckhoff_ER2xxx.Beckhoff_ER2xxxEK1122.A_0042_ER2349_0022_0017.Channel_24.Output <-> Channel 24/Output
//     PlcTask Outputs/GVL_iXlinker.EtherCAT_Master_ERxxxx.Beckhoff_ER2xxx.Beckhoff_ER2xxxEK1122.A_0042_ER2349_0022_0017.Channel_25.Output <-> Channel 25/Output
//     PlcTask Outputs/GVL_iXlinker.EtherCAT_Master_ERxxxx.Beckhoff_ER2xxx.Beckhoff_ER2xxxEK1122.A_0042_ER2349_0022_0017.Channel_26.Output <-> Channel 26/Output
//     PlcTask Outputs/GVL_iXlinker.EtherCAT_Master_ERxxxx.Beckhoff_ER2xxx.Beckhoff_ER2xxxEK1122.A_0042_ER2349_0022_0017.Channel_27.Output <-> Channel 27/Output
//     PlcTask Outputs/GVL_iXlinker.EtherCAT_Master_ERxxxx.Beckhoff_ER2xxx.Beckhoff_ER2xxxEK1122.A_0042_ER2349_0022_0017.Channel_28.Output <-> Channel 28/Output
//     PlcTask Outputs/GVL_iXlinker.EtherCAT_Master_ERxxxx.Beckhoff_ER2xxx.Beckhoff_ER2xxxEK1122.A_0042_ER2349_0022_0017.Channel_29.Output <-> Channel 29/Output
//     PlcTask Outputs/GVL_iXlinker.EtherCAT_Master_ERxxxx.Beckhoff_ER2xxx.Beckhoff_ER2xxxEK1122.A_0042_ER2349_0022_0017.Channel_30.Output <-> Channel 30/Output
//     PlcTask Outputs/GVL_iXlinker.EtherCAT_Master_ERxxxx.Beckhoff_ER2xxx.Beckhoff_ER2xxxEK1122.A_0042_ER2349_0022_0017.Channel_31.Output <-> Channel 31/Output
//     PlcTask Outputs/GVL_iXlinker.EtherCAT_Master_ERxxxx.Beckhoff_ER2xxx.Beckhoff_ER2xxxEK1122.A_0042_ER2349_0022_0017.Channel_32.Output <-> Channel 32/Output
//     PlcTask Inputs/GVL_iXlinker.EtherCAT_Master_ERxxxx.Beckhoff_ER2xxx.Beckhoff_ER2xxxEK1122.A_0042_ER2349_0022_0017.WcState.WcState <-> WcState/WcState
//     PlcTask Inputs/GVL_iXlinker.EtherCAT_Master_ERxxxx.Beckhoff_ER2xxx.Beckhoff_ER2xxxEK1122.A_0042_ER2349_0022_0017.WcState.InputToggle <-> WcState/InputToggle
//     PlcTask Inputs/GVL_iXlinker.EtherCAT_Master_ERxxxx.Beckhoff_ER2xxx.Beckhoff_ER2xxxEK1122.A_0042_ER2349_0022_0017.InfoData.State <-> InfoData/State
//   PLC/PLC Instance <-> EtherCAT Master ERxxxx/Beckhoff ER2xxx/Beckhoff ER2xxxEK1122/A_0043(ER2349-0022-0018)
//     PlcTask Inputs/GVL_iXlinker.EtherCAT_Master_ERxxxx.Beckhoff_ER2xxx.Beckhoff_ER2xxxEK1122.A_0043_ER2349_0022_0018.Channel_1.Input <-> Channel 1/Input
//     PlcTask Inputs/GVL_iXlinker.EtherCAT_Master_ERxxxx.Beckhoff_ER2xxx.Beckhoff_ER2xxxEK1122.A_0043_ER2349_0022_0018.Channel_2.Input <-> Channel 2/Input
//     PlcTask Inputs/GVL_iXlinker.EtherCAT_Master_ERxxxx.Beckhoff_ER2xxx.Beckhoff_ER2xxxEK1122.A_0043_ER2349_0022_0018.Channel_3.Input <-> Channel 3/Input
//     PlcTask Inputs/GVL_iXlinker.EtherCAT_Master_ERxxxx.Beckhoff_ER2xxx.Beckhoff_ER2xxxEK1122.A_0043_ER2349_0022_0018.Channel_4.Input <-> Channel 4/Input
//     PlcTask Inputs/GVL_iXlinker.EtherCAT_Master_ERxxxx.Beckhoff_ER2xxx.Beckhoff_ER2xxxEK1122.A_0043_ER2349_0022_0018.Channel_5.Input <-> Channel 5/Input
//     PlcTask Inputs/GVL_iXlinker.EtherCAT_Master_ERxxxx.Beckhoff_ER2xxx.Beckhoff_ER2xxxEK1122.A_0043_ER2349_0022_0018.Channel_6.Input <-> Channel 6/Input
//     PlcTask Inputs/GVL_iXlinker.EtherCAT_Master_ERxxxx.Beckhoff_ER2xxx.Beckhoff_ER2xxxEK1122.A_0043_ER2349_0022_0018.Channel_7.Input <-> Channel 7/Input
//     PlcTask Inputs/GVL_iXlinker.EtherCAT_Master_ERxxxx.Beckhoff_ER2xxx.Beckhoff_ER2xxxEK1122.A_0043_ER2349_0022_0018.Channel_8.Input <-> Channel 8/Input
//     PlcTask Inputs/GVL_iXlinker.EtherCAT_Master_ERxxxx.Beckhoff_ER2xxx.Beckhoff_ER2xxxEK1122.A_0043_ER2349_0022_0018.Channel_9.Input <-> Channel 9/Input
//     PlcTask Inputs/GVL_iXlinker.EtherCAT_Master_ERxxxx.Beckhoff_ER2xxx.Beckhoff_ER2xxxEK1122.A_0043_ER2349_0022_0018.Channel_10.Input <-> Channel 10/Input
//     PlcTask Inputs/GVL_iXlinker.EtherCAT_Master_ERxxxx.Beckhoff_ER2xxx.Beckhoff_ER2xxxEK1122.A_0043_ER2349_0022_0018.Channel_11.Input <-> Channel 11/Input
//     PlcTask Inputs/GVL_iXlinker.EtherCAT_Master_ERxxxx.Beckhoff_ER2xxx.Beckhoff_ER2xxxEK1122.A_0043_ER2349_0022_0018.Channel_12.Input <-> Channel 12/Input
//     PlcTask Inputs/GVL_iXlinker.EtherCAT_Master_ERxxxx.Beckhoff_ER2xxx.Beckhoff_ER2xxxEK1122.A_0043_ER2349_0022_0018.Channel_13.Input <-> Channel 13/Input
//     PlcTask Inputs/GVL_iXlinker.EtherCAT_Master_ERxxxx.Beckhoff_ER2xxx.Beckhoff_ER2xxxEK1122.A_0043_ER2349_0022_0018.Channel_14.Input <-> Channel 14/Input
//     PlcTask Inputs/GVL_iXlinker.EtherCAT_Master_ERxxxx.Beckhoff_ER2xxx.Beckhoff_ER2xxxEK1122.A_0043_ER2349_0022_0018.Channel_15.Input <-> Channel 15/Input
//     PlcTask Inputs/GVL_iXlinker.EtherCAT_Master_ERxxxx.Beckhoff_ER2xxx.Beckhoff_ER2xxxEK1122.A_0043_ER2349_0022_0018.Channel_16.Input <-> Channel 16/Input
//     PlcTask Outputs/GVL_iXlinker.EtherCAT_Master_ERxxxx.Beckhoff_ER2xxx.Beckhoff_ER2xxxEK1122.A_0043_ER2349_0022_0018.Channel_17.Output <-> Channel 17/Output
//     PlcTask Outputs/GVL_iXlinker.EtherCAT_Master_ERxxxx.Beckhoff_ER2xxx.Beckhoff_ER2xxxEK1122.A_0043_ER2349_0022_0018.Channel_18.Output <-> Channel 18/Output
//     PlcTask Outputs/GVL_iXlinker.EtherCAT_Master_ERxxxx.Beckhoff_ER2xxx.Beckhoff_ER2xxxEK1122.A_0043_ER2349_0022_0018.Channel_19.Output <-> Channel 19/Output
//     PlcTask Outputs/GVL_iXlinker.EtherCAT_Master_ERxxxx.Beckhoff_ER2xxx.Beckhoff_ER2xxxEK1122.A_0043_ER2349_0022_0018.Channel_20.Output <-> Channel 20/Output
//     PlcTask Outputs/GVL_iXlinker.EtherCAT_Master_ERxxxx.Beckhoff_ER2xxx.Beckhoff_ER2xxxEK1122.A_0043_ER2349_0022_0018.Channel_21.Output <-> Channel 21/Output
//     PlcTask Outputs/GVL_iXlinker.EtherCAT_Master_ERxxxx.Beckhoff_ER2xxx.Beckhoff_ER2xxxEK1122.A_0043_ER2349_0022_0018.Channel_22.Output <-> Channel 22/Output
//     PlcTask Outputs/GVL_iXlinker.EtherCAT_Master_ERxxxx.Beckhoff_ER2xxx.Beckhoff_ER2xxxEK1122.A_0043_ER2349_0022_0018.Channel_23.Output <-> Channel 23/Output
//     PlcTask Outputs/GVL_iXlinker.EtherCAT_Master_ERxxxx.Beckhoff_ER2xxx.Beckhoff_ER2xxxEK1122.A_0043_ER2349_0022_0018.Channel_24.Output <-> Channel 24/Output
//     PlcTask Outputs/GVL_iXlinker.EtherCAT_Master_ERxxxx.Beckhoff_ER2xxx.Beckhoff_ER2xxxEK1122.A_0043_ER2349_0022_0018.Channel_25.Output <-> Channel 25/Output
//     PlcTask Outputs/GVL_iXlinker.EtherCAT_Master_ERxxxx.Beckhoff_ER2xxx.Beckhoff_ER2xxxEK1122.A_0043_ER2349_0022_0018.Channel_26.Output <-> Channel 26/Output
//     PlcTask Outputs/GVL_iXlinker.EtherCAT_Master_ERxxxx.Beckhoff_ER2xxx.Beckhoff_ER2xxxEK1122.A_0043_ER2349_0022_0018.Channel_27.Output <-> Channel 27/Output
//     PlcTask Outputs/GVL_iXlinker.EtherCAT_Master_ERxxxx.Beckhoff_ER2xxx.Beckhoff_ER2xxxEK1122.A_0043_ER2349_0022_0018.Channel_28.Output <-> Channel 28/Output
//     PlcTask Outputs/GVL_iXlinker.EtherCAT_Master_ERxxxx.Beckhoff_ER2xxx.Beckhoff_ER2xxxEK1122.A_0043_ER2349_0022_0018.Channel_29.Output <-> Channel 29/Output
//     PlcTask Outputs/GVL_iXlinker.EtherCAT_Master_ERxxxx.Beckhoff_ER2xxx.Beckhoff_ER2xxxEK1122.A_0043_ER2349_0022_0018.Channel_30.Output <-> Channel 30/Output
//     PlcTask Outputs/GVL_iXlinker.EtherCAT_Master_ERxxxx.Beckhoff_ER2xxx.Beckhoff_ER2xxxEK1122.A_0043_ER2349_0022_0018.Channel_31.Output <-> Channel 31/Output
//     PlcTask Outputs/GVL_iXlinker.EtherCAT_Master_ERxxxx.Beckhoff_ER2xxx.Beckhoff_ER2xxxEK1122.A_0043_ER2349_0022_0018.Channel_32.Output <-> Channel 32/Output
//     PlcTask Inputs/GVL_iXlinker.EtherCAT_Master_ERxxxx.Beckhoff_ER2xxx.Beckhoff_ER2xxxEK1122.A_0043_ER2349_0022_0018.WcState.WcState <-> WcState/WcState
//     PlcTask Inputs/GVL_iXlinker.EtherCAT_Master_ERxxxx.Beckhoff_ER2xxx.Beckhoff_ER2xxxEK1122.A_0043_ER2349_0022_0018.WcState.InputToggle <-> WcState/InputToggle
//     PlcTask Inputs/GVL_iXlinker.EtherCAT_Master_ERxxxx.Beckhoff_ER2xxx.Beckhoff_ER2xxxEK1122.A_0043_ER2349_0022_0018.InfoData.State <-> InfoData/State
//   PLC/PLC Instance <-> EtherCAT Master ERxxxx/Beckhoff ER2xxx/Beckhoff ER2xxxEK1122/A_0044(ER2624-0002-0018)
//     PlcTask Outputs/GVL_iXlinker.EtherCAT_Master_ERxxxx.Beckhoff_ER2xxx.Beckhoff_ER2xxxEK1122.A_0044_ER2624_0002_0018.Channel_1.Output <-> Channel 1/Output
//     PlcTask Outputs/GVL_iXlinker.EtherCAT_Master_ERxxxx.Beckhoff_ER2xxx.Beckhoff_ER2xxxEK1122.A_0044_ER2624_0002_0018.Channel_2.Output <-> Channel 2/Output
//     PlcTask Outputs/GVL_iXlinker.EtherCAT_Master_ERxxxx.Beckhoff_ER2xxx.Beckhoff_ER2xxxEK1122.A_0044_ER2624_0002_0018.Channel_3.Output <-> Channel 3/Output
//     PlcTask Outputs/GVL_iXlinker.EtherCAT_Master_ERxxxx.Beckhoff_ER2xxx.Beckhoff_ER2xxxEK1122.A_0044_ER2624_0002_0018.Channel_4.Output <-> Channel 4/Output
//     PlcTask Inputs/GVL_iXlinker.EtherCAT_Master_ERxxxx.Beckhoff_ER2xxx.Beckhoff_ER2xxxEK1122.A_0044_ER2624_0002_0018.WcState.WcState <-> WcState/WcState
//     PlcTask Inputs/GVL_iXlinker.EtherCAT_Master_ERxxxx.Beckhoff_ER2xxx.Beckhoff_ER2xxxEK1122.A_0044_ER2624_0002_0018.InfoData.State <-> InfoData/State
//   PLC/PLC Instance <-> EtherCAT Master ERxxxx/Beckhoff ER2xxx/Beckhoff ER2xxxEK1122/A_0045(ER2624-0002-0019)
//     PlcTask Outputs/GVL_iXlinker.EtherCAT_Master_ERxxxx.Beckhoff_ER2xxx.Beckhoff_ER2xxxEK1122.A_0045_ER2624_0002_0019.Channel_1.Output <-> Channel 1/Output
//     PlcTask Outputs/GVL_iXlinker.EtherCAT_Master_ERxxxx.Beckhoff_ER2xxx.Beckhoff_ER2xxxEK1122.A_0045_ER2624_0002_0019.Channel_2.Output <-> Channel 2/Output
//     PlcTask Outputs/GVL_iXlinker.EtherCAT_Master_ERxxxx.Beckhoff_ER2xxx.Beckhoff_ER2xxxEK1122.A_0045_ER2624_0002_0019.Channel_3.Output <-> Channel 3/Output
//     PlcTask Outputs/GVL_iXlinker.EtherCAT_Master_ERxxxx.Beckhoff_ER2xxx.Beckhoff_ER2xxxEK1122.A_0045_ER2624_0002_0019.Channel_4.Output <-> Channel 4/Output
//     PlcTask Inputs/GVL_iXlinker.EtherCAT_Master_ERxxxx.Beckhoff_ER2xxx.Beckhoff_ER2xxxEK1122.A_0045_ER2624_0002_0019.WcState.WcState <-> WcState/WcState
//     PlcTask Inputs/GVL_iXlinker.EtherCAT_Master_ERxxxx.Beckhoff_ER2xxx.Beckhoff_ER2xxxEK1122.A_0045_ER2624_0002_0019.InfoData.State <-> InfoData/State
//   PLC/PLC Instance <-> EtherCAT Master ERxxxx/Beckhoff ER2xxx/Beckhoff ER2xxxEK1122/A_0046(ER2809-0021-0017)
//     PlcTask Outputs/GVL_iXlinker.EtherCAT_Master_ERxxxx.Beckhoff_ER2xxx.Beckhoff_ER2xxxEK1122.A_0046_ER2809_0021_0017.Channel_1.Output <-> Channel 1/Output
//     PlcTask Outputs/GVL_iXlinker.EtherCAT_Master_ERxxxx.Beckhoff_ER2xxx.Beckhoff_ER2xxxEK1122.A_0046_ER2809_0021_0017.Channel_2.Output <-> Channel 2/Output
//     PlcTask Outputs/GVL_iXlinker.EtherCAT_Master_ERxxxx.Beckhoff_ER2xxx.Beckhoff_ER2xxxEK1122.A_0046_ER2809_0021_0017.Channel_3.Output <-> Channel 3/Output
//     PlcTask Outputs/GVL_iXlinker.EtherCAT_Master_ERxxxx.Beckhoff_ER2xxx.Beckhoff_ER2xxxEK1122.A_0046_ER2809_0021_0017.Channel_4.Output <-> Channel 4/Output
//     PlcTask Outputs/GVL_iXlinker.EtherCAT_Master_ERxxxx.Beckhoff_ER2xxx.Beckhoff_ER2xxxEK1122.A_0046_ER2809_0021_0017.Channel_5.Output <-> Channel 5/Output
//     PlcTask Outputs/GVL_iXlinker.EtherCAT_Master_ERxxxx.Beckhoff_ER2xxx.Beckhoff_ER2xxxEK1122.A_0046_ER2809_0021_0017.Channel_6.Output <-> Channel 6/Output
//     PlcTask Outputs/GVL_iXlinker.EtherCAT_Master_ERxxxx.Beckhoff_ER2xxx.Beckhoff_ER2xxxEK1122.A_0046_ER2809_0021_0017.Channel_7.Output <-> Channel 7/Output
//     PlcTask Outputs/GVL_iXlinker.EtherCAT_Master_ERxxxx.Beckhoff_ER2xxx.Beckhoff_ER2xxxEK1122.A_0046_ER2809_0021_0017.Channel_8.Output <-> Channel 8/Output
//     PlcTask Outputs/GVL_iXlinker.EtherCAT_Master_ERxxxx.Beckhoff_ER2xxx.Beckhoff_ER2xxxEK1122.A_0046_ER2809_0021_0017.Channel_9.Output <-> Channel 9/Output
//     PlcTask Outputs/GVL_iXlinker.EtherCAT_Master_ERxxxx.Beckhoff_ER2xxx.Beckhoff_ER2xxxEK1122.A_0046_ER2809_0021_0017.Channel_10.Output <-> Channel 10/Output
//     PlcTask Outputs/GVL_iXlinker.EtherCAT_Master_ERxxxx.Beckhoff_ER2xxx.Beckhoff_ER2xxxEK1122.A_0046_ER2809_0021_0017.Channel_11.Output <-> Channel 11/Output
//     PlcTask Outputs/GVL_iXlinker.EtherCAT_Master_ERxxxx.Beckhoff_ER2xxx.Beckhoff_ER2xxxEK1122.A_0046_ER2809_0021_0017.Channel_12.Output <-> Channel 12/Output
//     PlcTask Outputs/GVL_iXlinker.EtherCAT_Master_ERxxxx.Beckhoff_ER2xxx.Beckhoff_ER2xxxEK1122.A_0046_ER2809_0021_0017.Channel_13.Output <-> Channel 13/Output
//     PlcTask Outputs/GVL_iXlinker.EtherCAT_Master_ERxxxx.Beckhoff_ER2xxx.Beckhoff_ER2xxxEK1122.A_0046_ER2809_0021_0017.Channel_14.Output <-> Channel 14/Output
//     PlcTask Outputs/GVL_iXlinker.EtherCAT_Master_ERxxxx.Beckhoff_ER2xxx.Beckhoff_ER2xxxEK1122.A_0046_ER2809_0021_0017.Channel_15.Output <-> Channel 15/Output
